LIN {X 0,Y 300.295,Z 456.079,A -85,B 0,C 180,E1 -16621.818,E2 -16621.818} C_VEL
LIN {X 0,Y 302.609,Z 468.728,A -85,B 0,C 180,E1 -16623.149,E2 -16623.149} C_VEL
LIN {X 0,Y 303.712,Z 478.266,A -85,B 0,C 180,E1 -16624.27,E2 -16624.27} C_VEL
LIN {X 0,Y 301.679,Z 491.184,A -85,B 0,C 180,E1 -16625.757,E2 -16625.757} C_VEL
LIN {X 0,Y 299.382,Z 502.708,A -85,B 0,C 180,E1 -16627.393,E2 -16627.393} C_VEL
LIN {X 0,Y 297.232,Z 513.15,A -85,B 0,C 180,E1 -16629.226,E2 -16629.226} C_VEL
LIN {X 0,Y 295.179,Z 522.585,A -85,B 0,C 180,E1 -16631.251,E2 -16631.251} C_VEL
LIN {X 0,Y 293.39,Z 531.306,A -85,B 0,C 180,E1 -16633.567,E2 -16633.567} C_VEL
LIN {X 0,Y 291.879,Z 538.835,A -85,B 0,C 180,E1 -16636.067,E2 -16636.067} C_VEL
LIN {X 0,Y 290.836,Z 543.926,A -85,B 0,C 180,E1 -16638.147,E2 -16638.147} C_VEL
LIN {X 0,Y 290.013,Z 549.179,A -85,B 0,C 180,E1 -16640.937,E2 -16640.937} C_VEL
LIN {X 0,Y 289.605,Z 552.122,A -85,B 0,C 180,E1 -16643.031,E2 -16643.031} C_VEL
LIN {X 0,Y 289.393,Z 554.815,A -85,B 0,C 180,E1 -16645.822,E2 -16645.822} C_VEL
LIN {X 0,Y 289.37,Z 556.148,A -85,B 0,C 180,E1 -16648.608,E2 -16648.608} C_VEL
LIN {X 0,Y 289.37,Z 556.142,A -85,B 0,C 180,E1 -16651.392,E2 -16651.392} C_VEL
LIN {X 0,Y 289.394,Z 554.801,A -85,B 0,C 180,E1 -16654.178,E2 -16654.178} C_VEL
LIN {X 0,Y 289.635,Z 552.099,A -85,B 0,C 180,E1 -16656.968,E2 -16656.968} C_VEL
LIN {X 0,Y 290.155,Z 547.96,A -85,B 0,C 180,E1 -16659.762,E2 -16659.762} C_VEL
LIN {X 0,Y 291.096,Z 542.261,A -85,B 0,C 180,E1 -16662.55,E2 -16662.55} C_VEL
LIN {X 0,Y 292.455,Z 535.839,A -85,B 0,C 180,E1 -16664.971,E2 -16664.971} C_VEL
LIN {X 0,Y 294.069,Z 527.863,A -85,B 0,C 180,E1 -16667.381,E2 -16667.381} C_VEL
LIN {X 0,Y 295.831,Z 519.513,A -85,B 0,C 180,E1 -16669.426,E2 -16669.426} C_VEL
LIN {X 0,Y 298.01,Z 509.466,A -85,B 0,C 180,E1 -16671.441,E2 -16671.441} C_VEL
LIN {X 0,Y 300.3,Z 498.252,A -85,B 0,C 180,E1 -16673.262,E2 -16673.262} C_VEL
LIN {X 0,Y 302.354,Z 487.095,A -85,B 0,C 180,E1 -16674.733,E2 -16674.733} C_VEL
LIN {X 0,Y 303.612,Z 477.752,A -85,B 0,C 180,E1 -16675.774,E2 -16675.774} C_VEL
LIN {X 0,Y 302.073,Z 465.248,A -85,B 0,C 180,E1 -16677.202,E2 -16677.202} C_VEL
LIN {X 0,Y 299.462,Z 452.518,A -85,B 0,C 180,E1 -16678.499,E2 -16678.499} C_VEL
LIN {X 0,Y 295.713,Z 438.551,A -85,B 0,C 180,E1 -16679.75,E2 -16679.75} C_VEL
LIN {X 0,Y 291.433,Z 426.246,A -85,B 0,C 180,E1 -16680.738,E2 -16680.738} C_VEL
LIN {X 0,Y 291.338,Z 425.398,A -85,B 0,C 180,E1 -16680.838,E2 -16680.838} C_VEL
LIN {X 0,Y 291.981,Z 420.382,A -85,B 0,C 180,E1 -16685.287,E2 -16685.287} C_VEL
LIN {X 0,Y 292.367,Z 416.77,A -85,B 0,C 180,E1 -16688.682,E2 -16688.682} C_VEL
LIN {X 0,Y 292.333,Z 413.602,A -85,B 0,C 180,E1 -16691.818,E2 -16691.818} C_VEL
LIN {X 0,Y 291.868,Z 409.987,A -85,B 0,C 180,E1 -16695.709,E2 -16695.709} C_VEL
LIN {X 0,Y 291.385,Z 406.828,A -85,B 0,C 180,E1 -16699.366,E2 -16699.366} C_VEL
LIN {X 0,Y 291.434,Z 406.81,A -85,B 0,C 180,E1 -16702.924,E2 -16702.924} C_VEL
LIN {X 0,Y 291.345,Z 406.822,A -85,B 0,C 180,E1 -16706.302,E2 -16706.302} C_VEL
LIN {X 0,Y 291.384,Z 406.816,A -85,B 0,C 180,E1 -16710.261,E2 -16710.261} C_VEL
LIN {X 0,Y 291.416,Z 406.812,A -85,B 0,C 180,E1 -16714.272,E2 -16714.272} C_VEL
LIN {X 0,Y 291.375,Z 406.817,A -85,B 0,C 180,E1 -16717.299,E2 -16717.299} C_VEL
LIN {X 0,Y 291.458,Z 406.805,A -85,B 0,C 180,E1 -16720.27,E2 -16720.27} C_VEL
LIN {X 0,Y 291.556,Z 406.792,A -85,B 0,C 180,E1 -16724.624,E2 -16724.624} C_VEL
LIN {X 0,Y 291.538,Z 406.791,A -85,B 0,C 180,E1 -16728.881,E2 -16728.881} C_VEL
LIN {X 0,Y 291.711,Z 406.773,A -85,B 0,C 180,E1 -16731.689,E2 -16731.689} C_VEL
LIN {X 0,Y 291.633,Z 406.783,A -85,B 0,C 180,E1 -16734.468,E2 -16734.468} C_VEL
LIN {X 0,Y 291.892,Z 406.753,A -85,B 0,C 180,E1 -16738.62,E2 -16738.62} C_VEL
LIN {X 0,Y 291.891,Z 406.752,A -85,B 0,C 180,E1 -16741.38,E2 -16741.38} C_VEL
LIN {X 0,Y 291.748,Z 406.769,A -85,B 0,C 180,E1 -16746.918,E2 -16746.918} C_VEL
LIN {X 0,Y 291.631,Z 406.786,A -85,B 0,C 180,E1 -16749.712,E2 -16749.712} C_VEL
LIN {X 0,Y 291.523,Z 406.792,A -85,B 0,C 180,E1 -16753.95,E2 -16753.95} C_VEL
LIN {X 0,Y 291.489,Z 406.796,A -85,B 0,C 180,E1 -16756.818,E2 -16756.818} C_VEL
LIN {X 0,Y 291.452,Z 406.806,A -85,B 0,C 180,E1 -16759.875,E2 -16759.875} C_VEL
LIN {X 0,Y 291.401,Z 406.813,A -85,B 0,C 180,E1 -16764.205,E2 -16764.205} C_VEL
LIN {X 0,Y 291.422,Z 406.81,A -85,B 0,C 180,E1 -16767.272,E2 -16767.272} C_VEL
LIN {X 0,Y 291.335,Z 406.82,A -85,B 0,C 180,E1 -16770.437,E2 -16770.437} C_VEL
LIN {X 0,Y 291.346,Z 406.82,A -85,B 0,C 180,E1 -16773.698,E2 -16773.698} C_VEL
LIN {X 0,Y 291.396,Z 406.815,A -85,B 0,C 180,E1 -16777.259,E2 -16777.259} C_VEL
LIN {X 0,Y 291.335,Z 406.823,A -85,B 0,C 180,E1 -16780.642,E2 -16780.642} C_VEL
LIN {X 0,Y 291.328,Z 406.82,A -85,B 0,C 180,E1 -16783.637,E2 -16783.637} C_VEL
LIN {X 0,Y 291.766,Z 409.919,A -85,B 0,C 180,E1 -16787.588,E2 -16787.588} C_VEL
LIN {X 0,Y 291.906,Z 412.394,A -85,B 0,C 180,E1 -16790.394,E2 -16790.394} C_VEL
LIN {X 0,Y 291.817,Z 414.778,A -85,B 0,C 180,E1 -16792.98,E2 -16792.98} C_VEL
LIN {X 0,Y 291.499,Z 417.991,A -85,B 0,C 180,E1 -16796.322,E2 -16796.322} C_VEL
LIN {X 0,Y 291.169,Z 420.912,A -85,B 0,C 180,E1 -16799.241,E2 -16799.241} C_VEL
LIN {X 0,Y 292.268,Z 424.311,A -85,B 0,C 180,E1 -16799.502,E2 -16799.502} C_VEL
LIN {X 0,Y 297.035,Z 437.696,A -85,B 0,C 180,E1 -16800.662,E2 -16800.662} C_VEL
LIN {X 0,Y 300.646,Z 451.139,A -85,B 0,C 180,E1 -16801.942,E2 -16801.942} C_VEL
LIN {X 0,Y 303.006,Z 462.696,A -85,B 0,C 180,E1 -16803.185,E2 -16803.185} C_VEL
LIN {X 0,Y 304.162,Z 470.973,A -85,B 0,C 180,E1 -16804.15,E2 -16804.15} C_VEL
LIN {X 0,Y 302.788,Z 481.413,A -85,B 0,C 180,E1 -16805.305,E2 -16805.305} C_VEL
LIN {X 0,Y 300.717,Z 492.606,A -85,B 0,C 180,E1 -16806.773,E2 -16806.773} C_VEL
LIN {X 0,Y 298.355,Z 503.859,A -85,B 0,C 180,E1 -16808.585,E2 -16808.585} C_VEL
LIN {X 0,Y 296.208,Z 513.912,A -85,B 0,C 180,E1 -16810.599,E2 -16810.599} C_VEL
LIN {X 0,Y 294.184,Z 523.069,A -85,B 0,C 180,E1 -16812.862,E2 -16812.862} C_VEL
LIN {X 0,Y 292.864,Z 530.227,A -85,B 0,C 180,E1 -16815.05,E2 -16815.05} C_VEL
LIN {X 0,Y 291.379,Z 536.643,A -85,B 0,C 180,E1 -16817.463,E2 -16817.463} C_VEL
LIN {X 0,Y 290.364,Z 542.331,A -85,B 0,C 180,E1 -16820.246,E2 -16820.246} C_VEL
LIN {X 0,Y 289.775,Z 546.463,A -85,B 0,C 180,E1 -16823.035,E2 -16823.035} C_VEL
LIN {X 0,Y 289.481,Z 549.164,A -85,B 0,C 180,E1 -16825.823,E2 -16825.823} C_VEL
LIN {X 0,Y 289.384,Z 550.516,A -85,B 0,C 180,E1 -16828.609,E2 -16828.609} C_VEL
LIN {X 0,Y 289.383,Z 550.546,A -85,B 0,C 180,E1 -16831.392,E2 -16831.392} C_VEL
LIN {X 0,Y 289.48,Z 549.251,A -85,B 0,C 180,E1 -16834.177,E2 -16834.177} C_VEL
LIN {X 0,Y 289.774,Z 546.601,A -85,B 0,C 180,E1 -16836.965,E2 -16836.965} C_VEL
LIN {X 0,Y 290.348,Z 542.528,A -85,B 0,C 180,E1 -16839.755,E2 -16839.755} C_VEL
LIN {X 0,Y 291.351,Z 536.901,A -85,B 0,C 180,E1 -16842.539,E2 -16842.539} C_VEL
LIN {X 0,Y 292.822,Z 530.546,A -85,B 0,C 180,E1 -16844.952,E2 -16844.952} C_VEL
LIN {X 0,Y 294.402,Z 522.572,A -85,B 0,C 180,E1 -16847.384,E2 -16847.384} C_VEL
LIN {X 0,Y 296.171,Z 514.38,A -85,B 0,C 180,E1 -16849.403,E2 -16849.403} C_VEL
LIN {X 0,Y 298.315,Z 504.42,A -85,B 0,C 180,E1 -16851.418,E2 -16851.418} C_VEL
LIN {X 0,Y 300.625,Z 493.329,A -85,B 0,C 180,E1 -16853.235,E2 -16853.235} C_VEL
LIN {X 0,Y 302.888,Z 480.905,A -85,B 0,C 180,E1 -16854.867,E2 -16854.867} C_VEL
LIN {X 0,Y 304.238,Z 471.314,A -85,B 0,C 180,E1 -16855.918,E2 -16855.918} C_VEL
LIN {X 0,Y 302.444,Z 459.661,A -85,B 0,C 180,E1 -16857.273,E2 -16857.273} C_VEL
LIN {X 0,Y 299.411,Z 446.078,A -85,B 0,C 180,E1 -16858.677,E2 -16858.677} C_VEL
LIN {X 0,Y 295.835,Z 433.958,A -85,B 0,C 180,E1 -16859.791,E2 -16859.791} C_VEL
LIN {X 0,Y 291.248,Z 421.639,A -85,B 0,C 180,E1 -16860.828,E2 -16860.828} C_VEL
LIN {X 0,Y 291.129,Z 420.907,A -85,B 0,C 180,E1 -16860.89,E2 -16860.89} C_VEL
LIN {X 0,Y 291.653,Z 416.829,A -85,B 0,C 180,E1 -16864.985,E2 -16864.985} C_VEL
LIN {X 0,Y 291.882,Z 413.257,A -85,B 0,C 180,E1 -16868.758,E2 -16868.758} C_VEL
LIN {X 0,Y 291.856,Z 410.636,A -85,B 0,C 180,E1 -16871.712,E2 -16871.712} C_VEL
LIN {X 0,Y 291.416,Z 407.395,A -85,B 0,C 180,E1 -16875.622,E2 -16875.622} C_VEL
LIN {X 0,Y 291.337,Z 406.828,A -85,B 0,C 180,E1 -16876.361,E2 -16876.361} C_VEL
LIN {X 0,Y 291.383,Z 406.815,A -85,B 0,C 180,E1 -16880.518,E2 -16880.518} C_VEL
LIN {X 0,Y 291.41,Z 406.813,A -85,B 0,C 180,E1 -16882.92,E2 -16882.92} C_VEL
LIN {X 0,Y 291.347,Z 406.82,A -85,B 0,C 180,E1 -16886.302,E2 -16886.302} C_VEL
LIN {X 0,Y 291.389,Z 406.812,A -85,B 0,C 180,E1 -16890.26,E2 -16890.26} C_VEL
LIN {X 0,Y 291.419,Z 406.811,A -85,B 0,C 180,E1 -16894.272,E2 -16894.272} C_VEL
LIN {X 0,Y 291.384,Z 406.814,A -85,B 0,C 180,E1 -16897.3,E2 -16897.3} C_VEL
LIN {X 0,Y 291.461,Z 406.8,A -85,B 0,C 180,E1 -16900.27,E2 -16900.27} C_VEL
LIN {X 0,Y 291.558,Z 406.791,A -85,B 0,C 180,E1 -16904.624,E2 -16904.624} C_VEL
LIN {X 0,Y 291.54,Z 406.795,A -85,B 0,C 180,E1 -16908.881,E2 -16908.881} C_VEL
LIN {X 0,Y 291.712,Z 406.772,A -85,B 0,C 180,E1 -16911.688,E2 -16911.688} C_VEL
LIN {X 0,Y 291.634,Z 406.783,A -85,B 0,C 180,E1 -16914.468,E2 -16914.468} C_VEL
LIN {X 0,Y 291.601,Z 406.783,A -85,B 0,C 180,E1 -16916.223,E2 -16916.223} C_VEL
LIN {X 0,Y 291.077,Z 406.853,A -85,B 0,C 180,E1 -16917.379,E2 -16917.379} C_VEL
LIN {X 0,Y 288.348,Z 407.192,A -85,B 0,C 180,E1 -16919.264,E2 -16919.264} C_VEL
LIN {X 0,Y 285.936,Z 407.49,A -85,B 0,C 180,E1 -16920.794,E2 -16920.794} C_VEL
LIN {X 0,Y 284.866,Z 407.627,A -85,B 0,C 180,E1 -16921.978,E2 -16921.978} C_VEL
LIN {X 0,Y 284.764,Z 407.636,A -85,B 0,C 180,E1 -16922.379,E2 -16922.379} C_VEL
LIN {X 0,Y 284.701,Z 407.646,A -85,B 0,C 180,E1 -16927.09,E2 -16927.09} C_VEL
LIN {X 0,Y 284.569,Z 407.663,A -85,B 0,C 180,E1 -16929.955,E2 -16929.955} C_VEL
LIN {X 0,Y 284.484,Z 407.675,A -85,B 0,C 180,E1 -16934.303,E2 -16934.303} C_VEL
LIN {X 0,Y 284.428,Z 407.679,A -85,B 0,C 180,E1 -16937.248,E2 -16937.248} C_VEL
LIN {X 0,Y 284.381,Z 407.687,A -85,B 0,C 180,E1 -16940.242,E2 -16940.242} C_VEL
LIN {X 0,Y 284.371,Z 407.682,A -85,B 0,C 180,E1 -16943.875,E2 -16943.875} C_VEL
LIN {X 0,Y 284.397,Z 407.68,A -85,B 0,C 180,E1 -16947.173,E2 -16947.173} C_VEL
LIN {X 0,Y 284.296,Z 407.698,A -85,B 0,C 180,E1 -16951.274,E2 -16951.274} C_VEL
LIN {X 0,Y 284.364,Z 407.692,A -85,B 0,C 180,E1 -16955.354,E2 -16955.354} C_VEL
LIN {X 0,Y 284.336,Z 407.697,A -85,B 0,C 180,E1 -16958.165,E2 -16958.165} C_VEL
LIN {X 0,Y 284.353,Z 407.696,A -85,B 0,C 180,E1 -16959.987,E2 -16959.987} C_VEL
LIN {X 0,Y 284.834,Z 410.735,A -85,B 0,C 180,E1 -16963.699,E2 -16963.699} C_VEL
LIN {X 0,Y 285.3,Z 414.29,A -85,B 0,C 180,E1 -16967.647,E2 -16967.647} C_VEL
LIN {X 0,Y 285.408,Z 416.721,A -85,B 0,C 180,E1 -16970.19,E2 -16970.19} C_VEL
LIN {X 0,Y 285.08,Z 420.364,A -85,B 0,C 180,E1 -16973.724,E2 -16973.724} C_VEL
LIN {X 0,Y 284.462,Z 424.903,A -85,B 0,C 180,E1 -16977.913,E2 -16977.913} C_VEL
LIN {X 0,Y 284.389,Z 425.386,A -85,B 0,C 180,E1 -16978.347,E2 -16978.347} C_VEL
LIN {X 0,Y 285.345,Z 428.635,A -85,B 0,C 180,E1 -16978.584,E2 -16978.584} C_VEL
LIN {X 0,Y 290.093,Z 442.311,A -85,B 0,C 180,E1 -16979.792,E2 -16979.792} C_VEL
LIN {X 0,Y 293.548,Z 456.013,A -85,B 0,C 180,E1 -16981.11,E2 -16981.11} C_VEL
LIN {X 0,Y 295.849,Z 468.661,A -85,B 0,C 180,E1 -16982.484,E2 -16982.484} C_VEL
LIN {X 0,Y 297.074,Z 480.142,A -85,B 0,C 180,E1 -16983.883,E2 -16983.883} C_VEL
LIN {X 0,Y 294.967,Z 492.411,A -85,B 0,C 180,E1 -16985.357,E2 -16985.357} C_VEL
LIN {X 0,Y 292.608,Z 503.706,A -85,B 0,C 180,E1 -16987.027,E2 -16987.027} C_VEL
LIN {X 0,Y 290.195,Z 514.769,A -85,B 0,C 180,E1 -16989.07,E2 -16989.07} C_VEL
LIN {X 0,Y 288.107,Z 523.897,A -85,B 0,C 180,E1 -16991.142,E2 -16991.142} C_VEL
LIN {X 0,Y 286.528,Z 530.915,A -85,B 0,C 180,E1 -16993.057,E2 -16993.057} C_VEL
LIN {X 0,Y 285.382,Z 536.846,A -85,B 0,C 180,E1 -16995.014,E2 -16995.014} C_VEL
LIN {X 0,Y 284.142,Z 542.246,A -85,B 0,C 180,E1 -16997.138,E2 -16997.138} C_VEL
LIN {X 0,Y 283.145,Z 547.93,A -85,B 0,C 180,E1 -16999.994,E2 -16999.994} C_VEL
LIN {X 0,Y 282.552,Z 552.054,A -85,B 0,C 180,E1 -17002.856,E2 -17002.856} C_VEL
LIN {X 0,Y 282.304,Z 554.747,A -85,B 0,C 180,E1 -17005.717,E2 -17005.717} C_VEL
LIN {X 0,Y 282.295,Z 556.079,A -85,B 0,C 180,E1 -17008.573,E2 -17008.573} C_VEL
LIN {X 0,Y 282.295,Z 556.074,A -85,B 0,C 180,E1 -17011.426,E2 -17011.426} C_VEL
LIN {X 0,Y 282.305,Z 554.732,A -85,B 0,C 180,E1 -17014.283,E2 -17014.283} C_VEL
LIN {X 0,Y 282.572,Z 552.03,A -85,B 0,C 180,E1 -17017.144,E2 -17017.144} C_VEL
LIN {X 0,Y 283.131,Z 547.89,A -85,B 0,C 180,E1 -17020.006,E2 -17020.006} C_VEL
LIN {X 0,Y 284.14,Z 542.191,A -85,B 0,C 180,E1 -17022.862,E2 -17022.862} C_VEL
LIN {X 0,Y 285.528,Z 535.768,A -85,B 0,C 180,E1 -17025.343,E2 -17025.343} C_VEL
LIN {X 0,Y 287.248,Z 527.789,A -85,B 0,C 180,E1 -17027.808,E2 -17027.808} C_VEL
LIN {X 0,Y 289.127,Z 519.442,A -85,B 0,C 180,E1 -17029.895,E2 -17029.895} C_VEL
LIN {X 0,Y 291.365,Z 509.394,A -85,B 0,C 180,E1 -17031.955,E2 -17031.955} C_VEL
LIN {X 0,Y 293.767,Z 498.179,A -85,B 0,C 180,E1 -17033.81,E2 -17033.81} C_VEL
LIN {X 0,Y 295.899,Z 487.022,A -85,B 0,C 180,E1 -17035.31,E2 -17035.31} C_VEL
LIN {X 0,Y 297.035,Z 479.43,A -85,B 0,C 180,E1 -17036.179,E2 -17036.179} C_VEL
LIN {X 0,Y 295.657,Z 467.162,A -85,B 0,C 180,E1 -17037.651,E2 -17037.651} C_VEL
LIN {X 0,Y 292.984,Z 453.827,A -85,B 0,C 180,E1 -17039.084,E2 -17039.084} C_VEL
LIN {X 0,Y 289.542,Z 440.775,A -85,B 0,C 180,E1 -17040.323,E2 -17040.323} C_VEL
LIN {X 0,Y 285.13,Z 428.161,A -85,B 0,C 180,E1 -17041.425,E2 -17041.425} C_VEL
LIN {X 0,Y 284.377,Z 425.375,A -85,B 0,C 180,E1 -17041.628,E2 -17041.628} C_VEL
LIN {X 0,Y 284.981,Z 421.125,A -85,B 0,C 180,E1 -17045.529,E2 -17045.529} C_VEL
LIN {X 0,Y 285.289,Z 418.511,A -85,B 0,C 180,E1 -17048.015,E2 -17048.015} C_VEL
LIN {X 0,Y 285.387,Z 416.271,A -85,B 0,C 180,E1 -17050.234,E2 -17050.234} C_VEL
LIN {X 0,Y 285.14,Z 413.066,A -85,B 0,C 180,E1 -17053.641,E2 -17053.641} C_VEL
LIN {X 0,Y 284.628,Z 409.423,A -85,B 0,C 180,E1 -17057.796,E2 -17057.796} C_VEL
LIN {X 0,Y 284.352,Z 407.693,A -85,B 0,C 180,E1 -17060.013,E2 -17060.013} C_VEL
LIN {X 0,Y 284.356,Z 407.691,A -85,B 0,C 180,E1 -17063.618,E2 -17063.618} C_VEL
LIN {X 0,Y 284.308,Z 407.698,A -85,B 0,C 180,E1 -17067.19,E2 -17067.19} C_VEL
LIN {X 0,Y 284.356,Z 407.692,A -85,B 0,C 180,E1 -17070.376,E2 -17070.376} C_VEL
LIN {X 0,Y 284.378,Z 407.688,A -85,B 0,C 180,E1 -17073.587,E2 -17073.587} C_VEL
LIN {X 0,Y 284.334,Z 407.693,A -85,B 0,C 180,E1 -17076.704,E2 -17076.704} C_VEL
LIN {X 0,Y 284.404,Z 407.683,A -85,B 0,C 180,E1 -17081.262,E2 -17081.262} C_VEL
LIN {X 0,Y 284.493,Z 407.672,A -85,B 0,C 180,E1 -17084.459,E2 -17084.459} C_VEL
LIN {X 0,Y 284.49,Z 407.669,A -85,B 0,C 180,E1 -17088.602,E2 -17088.602} C_VEL
LIN {X 0,Y 284.661,Z 407.652,A -85,B 0,C 180,E1 -17091.481,E2 -17091.481} C_VEL
LIN {X 0,Y 284.603,Z 407.658,A -85,B 0,C 180,E1 -17094.331,E2 -17094.331} C_VEL
LIN {X 0,Y 284.857,Z 407.629,A -85,B 0,C 180,E1 -17098.586,E2 -17098.586} C_VEL
LIN {X 0,Y 284.857,Z 407.629,A -85,B 0,C 180,E1 -17101.414,E2 -17101.414} C_VEL
LIN {X 0,Y 284.7,Z 407.647,A -85,B 0,C 180,E1 -17107.09,E2 -17107.09} C_VEL
LIN {X 0,Y 284.568,Z 407.663,A -85,B 0,C 180,E1 -17109.955,E2 -17109.955} C_VEL
LIN {X 0,Y 284.483,Z 407.67,A -85,B 0,C 180,E1 -17114.303,E2 -17114.303} C_VEL
LIN {X 0,Y 284.427,Z 407.676,A -85,B 0,C 180,E1 -17117.248,E2 -17117.248} C_VEL
LIN {X 0,Y 284.38,Z 407.686,A -85,B 0,C 180,E1 -17120.242,E2 -17120.242} C_VEL
LIN {X 0,Y 284.37,Z 407.688,A -85,B 0,C 180,E1 -17123.876,E2 -17123.876} C_VEL
LIN {X 0,Y 284.397,Z 407.685,A -85,B 0,C 180,E1 -17127.173,E2 -17127.173} C_VEL
LIN {X 0,Y 284.295,Z 407.698,A -85,B 0,C 180,E1 -17131.275,E2 -17131.275} C_VEL
LIN {X 0,Y 284.363,Z 407.69,A -85,B 0,C 180,E1 -17135.354,E2 -17135.354} C_VEL
LIN {X 0,Y 284.324,Z 407.692,A -85,B 0,C 180,E1 -17138.167,E2 -17138.167} C_VEL
LIN {X 0,Y 284.27,Z 407.702,A -85,B 0,C 180,E1 -17142.125,E2 -17142.125} C_VEL
LIN {X 0,Y 284.375,Z 408.375,A -85,B 0,C 180,E1 -17144.217,E2 -17144.217} C_VEL
LIN {X 0,Y 284.86,Z 411.602,A -85,B 0,C 180,E1 -17148.23,E2 -17148.23} C_VEL
LIN {X 0,Y 284.83,Z 414.853,A -85,B 0,C 180,E1 -17151.913,E2 -17151.913} C_VEL
LIN {X 0,Y 284.558,Z 418.073,A -85,B 0,C 180,E1 -17155.386,E2 -17155.386} C_VEL
LIN {X 0,Y 284.227,Z 421.003,A -85,B 0,C 180,E1 -17158.416,E2 -17158.416} C_VEL
LIN {X 0,Y 285.22,Z 424.218,A -85,B 0,C 180,E1 -17158.658,E2 -17158.658} C_VEL
LIN {X 0,Y 290.073,Z 437.415,A -85,B 0,C 180,E1 -17159.865,E2 -17159.865} C_VEL
LIN {X 0,Y 293.876,Z 451.158,A -85,B 0,C 180,E1 -17161.231,E2 -17161.231} C_VEL
LIN {X 0,Y 296.453,Z 463.855,A -85,B 0,C 180,E1 -17162.647,E2 -17162.647} C_VEL
LIN {X 0,Y 297.595,Z 473.419,A -85,B 0,C 180,E1 -17163.82,E2 -17163.82} C_VEL
LIN {X 0,Y 295.605,Z 485.426,A -85,B 0,C 180,E1 -17165.227,E2 -17165.227} C_VEL
LIN {X 0,Y 293.256,Z 497.006,A -85,B 0,C 180,E1 -17166.894,E2 -17166.894} C_VEL
LIN {X 0,Y 291.005,Z 507.488,A -85,B 0,C 180,E1 -17168.761,E2 -17168.761} C_VEL
LIN {X 0,Y 288.832,Z 516.948,A -85,B 0,C 180,E1 -17170.823,E2 -17170.823} C_VEL
LIN {X 0,Y 286.817,Z 525.968,A -85,B 0,C 180,E1 -17173.267,E2 -17173.267} C_VEL
LIN {X 0,Y 285.733,Z 531.302,A -85,B 0,C 180,E1 -17175.033,E2 -17175.033} C_VEL
LIN {X 0,Y 284.416,Z 536.714,A -85,B 0,C 180,E1 -17177.151,E2 -17177.151} C_VEL
LIN {X 0,Y 283.351,Z 542.401,A -85,B 0,C 180,E1 -17180.002,E2 -17180.002} C_VEL
LIN {X 0,Y 282.726,Z 546.533,A -85,B 0,C 180,E1 -17182.86,E2 -17182.86} C_VEL
LIN {X 0,Y 282.392,Z 549.234,A -85,B 0,C 180,E1 -17185.718,E2 -17185.718} C_VEL
LIN {X 0,Y 282.309,Z 550.585,A -85,B 0,C 180,E1 -17188.574,E2 -17188.574} C_VEL
LIN {X 0,Y 282.309,Z 550.614,A -85,B 0,C 180,E1 -17191.427,E2 -17191.427} C_VEL
LIN {X 0,Y 282.391,Z 549.319,A -85,B 0,C 180,E1 -17194.282,E2 -17194.282} C_VEL
LIN {X 0,Y 282.726,Z 546.669,A -85,B 0,C 180,E1 -17197.14,E2 -17197.14} C_VEL
LIN {X 0,Y 283.333,Z 542.596,A -85,B 0,C 180,E1 -17199.999,E2 -17199.999} C_VEL
LIN {X 0,Y 284.389,Z 536.969,A -85,B 0,C 180,E1 -17202.851,E2 -17202.851} C_VEL
LIN {X 0,Y 285.947,Z 530.613,A -85,B 0,C 180,E1 -17205.32,E2 -17205.32} C_VEL
LIN {X 0,Y 287.581,Z 522.695,A -85,B 0,C 180,E1 -17207.793,E2 -17207.793} C_VEL
LIN {X 0,Y 289.449,Z 514.447,A -85,B 0,C 180,E1 -17209.873,E2 -17209.873} C_VEL
LIN {X 0,Y 291.718,Z 504.485,A -85,B 0,C 180,E1 -17211.927,E2 -17211.927} C_VEL
LIN {X 0,Y 294.1,Z 493.394,A -85,B 0,C 180,E1 -17213.782,E2 -17213.782} C_VEL
LIN {X 0,Y 296.22,Z 482.35,A -85,B 0,C 180,E1 -17215.281,E2 -17215.281} C_VEL
LIN {X 0,Y 297.691,Z 472.69,A -85,B 0,C 180,E1 -17216.375,E2 -17216.375} C_VEL
LIN {X 0,Y 295.938,Z 461.06,A -85,B 0,C 180,E1 -17217.795,E2 -17217.795} C_VEL
LIN {X 0,Y 293.151,Z 448.192,A -85,B 0,C 180,E1 -17219.193,E2 -17219.193} C_VEL
LIN {X 0,Y 289.954,Z 437.068,A -85,B 0,C 180,E1 -17220.29,E2 -17220.29} C_VEL
LIN {X 0,Y 284.966,Z 423.701,A -85,B 0,C 180,E1 -17221.515,E2 -17221.515} C_VEL
LIN {X 0,Y 284.222,Z 420.978,A -85,B 0,C 180,E1 -17221.732,E2 -17221.732} C_VEL
LIN {X 0,Y 284.65,Z 417.399,A -85,B 0,C 180,E1 -17225.435,E2 -17225.435} C_VEL
LIN {X 0,Y 284.83,Z 414.949,A -85,B 0,C 180,E1 -17228.087,E2 -17228.087} C_VEL
LIN {X 0,Y 284.9,Z 413.145,A -85,B 0,C 180,E1 -17230.118,E2 -17230.118} C_VEL
LIN {X 0,Y 284.794,Z 411.328,A -85,B 0,C 180,E1 -17232.241,E2 -17232.241} C_VEL
LIN {X 0,Y 284.354,Z 408.153,A -85,B 0,C 180,E1 -17236.208,E2 -17236.208} C_VEL
LIN {X 0,Y 284.274,Z 407.705,A -85,B 0,C 180,E1 -17238.125,E2 -17238.125} C_VEL
LIN {X 0,Y 284.325,Z 407.693,A -85,B 0,C 180,E1 -17242.278,E2 -17242.278} C_VEL
LIN {X 0,Y 284.311,Z 407.696,A -85,B 0,C 180,E1 -17245.351,E2 -17245.351} C_VEL
LIN {X 0,Y 284.298,Z 407.696,A -85,B 0,C 180,E1 -17248.726,E2 -17248.726} C_VEL
LIN {X 0,Y 284.4,Z 407.686,A -85,B 0,C 180,E1 -17252.826,E2 -17252.826} C_VEL
LIN {X 0,Y 284.369,Z 407.684,A -85,B 0,C 180,E1 -17256.707,E2 -17256.707} C_VEL
LIN {X 0,Y 284.407,Z 407.683,A -85,B 0,C 180,E1 -17261.262,E2 -17261.262} C_VEL
LIN {X 0,Y 284.495,Z 407.671,A -85,B 0,C 180,E1 -17264.459,E2 -17264.459} C_VEL
LIN {X 0,Y 284.491,Z 407.673,A -85,B 0,C 180,E1 -17268.601,E2 -17268.601} C_VEL
LIN {X 0,Y 284.662,Z 407.65,A -85,B 0,C 180,E1 -17271.481,E2 -17271.481} C_VEL
LIN {X 0,Y 284.604,Z 407.658,A -85,B 0,C 180,E1 -17274.331,E2 -17274.331} C_VEL
LIN {X 0,Y 284.857,Z 407.627,A -85,B 0,C 180,E1 -17278.586,E2 -17278.586} C_VEL
LIN {X 0,Y 284.859,Z 407.626,A -85,B 0,C 180,E1 -17281.414,E2 -17281.414} C_VEL
LIN {X 0,Y 284.764,Z 407.636,A -85,B 0,C 180,E1 -17282.379,E2 -17282.379} C_VEL
LIN {X 0,Y 284.044,Z 407.729,A -85,B 0,C 180,E1 -17283.558,E2 -17283.558} C_VEL
LIN {X 0,Y 281.132,Z 408.089,A -85,B 0,C 180,E1 -17285.478,E2 -17285.478} C_VEL
LIN {X 0,Y 278.703,Z 408.394,A -85,B 0,C 180,E1 -17287.036,E2 -17287.036} C_VEL
LIN {X 0,Y 277.686,Z 408.52,A -85,B 0,C 180,E1 -17288.245,E2 -17288.245} C_VEL
LIN {X 0,Y 277.616,Z 408.529,A -85,B 0,C 180,E1 -17288.655,E2 -17288.655} C_VEL
LIN {X 0,Y 277.42,Z 408.555,A -85,B 0,C 180,E1 -17293.179,E2 -17293.179} C_VEL
LIN {X 0,Y 277.409,Z 408.557,A -85,B 0,C 180,E1 -17296.181,E2 -17296.181} C_VEL
LIN {X 0,Y 277.347,Z 408.563,A -85,B 0,C 180,E1 -17300.35,E2 -17300.35} C_VEL
LIN {X 0,Y 277.321,Z 408.56,A -85,B 0,C 180,E1 -17304.17,E2 -17304.17} C_VEL
LIN {X 0,Y 277.325,Z 408.561,A -85,B 0,C 180,E1 -17307.504,E2 -17307.504} C_VEL
LIN {X 0,Y 277.274,Z 408.569,A -85,B 0,C 180,E1 -17310.481,E2 -17310.481} C_VEL
LIN {X 0,Y 277.256,Z 408.577,A -85,B 0,C 180,E1 -17313.894,E2 -17313.894} C_VEL
LIN {X 0,Y 277.292,Z 408.575,A -85,B 0,C 180,E1 -17317.465,E2 -17317.465} C_VEL
LIN {X 0,Y 277.269,Z 408.578,A -85,B 0,C 180,E1 -17319.322,E2 -17319.322} C_VEL
LIN {X 0,Y 277.761,Z 411.472,A -85,B 0,C 180,E1 -17323.091,E2 -17323.091} C_VEL
LIN {X 0,Y 278.237,Z 414.928,A -85,B 0,C 180,E1 -17327.097,E2 -17327.097} C_VEL
LIN {X 0,Y 278.352,Z 416.929,A -85,B 0,C 180,E1 -17329.24,E2 -17329.24} C_VEL
LIN {X 0,Y 278.153,Z 420.281,A -85,B 0,C 180,E1 -17332.67,E2 -17332.67} C_VEL
LIN {X 0,Y 277.647,Z 423.925,A -85,B 0,C 180,E1 -17336.159,E2 -17336.159} C_VEL
LIN {X 0,Y 277.48,Z 425.306,A -85,B 0,C 180,E1 -17337.457,E2 -17337.457} C_VEL
LIN {X 0,Y 278.453,Z 428.552,A -85,B 0,C 180,E1 -17337.712,E2 -17337.712} C_VEL
LIN {X 0,Y 282.652,Z 440.529,A -85,B 0,C 180,E1 -17338.813,E2 -17338.813} C_VEL
LIN {X 0,Y 285.635,Z 451.022,A -85,B 0,C 180,E1 -17339.847,E2 -17339.847} C_VEL
LIN {X 0,Y 288.458,Z 464.356,A -85,B 0,C 180,E1 -17341.295,E2 -17341.295} C_VEL
LIN {X 0,Y 290.007,Z 475.033,A -85,B 0,C 180,E1 -17342.584,E2 -17342.584} C_VEL
LIN {X 0,Y 290.497,Z 481.435,A -85,B 0,C 180,E1 -17343.413,E2 -17343.413} C_VEL
LIN {X 0,Y 288.267,Z 493.58,A -85,B 0,C 180,E1 -17344.937,E2 -17344.937} C_VEL
LIN {X 0,Y 286.053,Z 503.64,A -85,B 0,C 180,E1 -17346.469,E2 -17346.469} C_VEL
LIN {X 0,Y 283.537,Z 514.702,A -85,B 0,C 180,E1 -17348.555,E2 -17348.555} C_VEL
LIN {X 0,Y 281.374,Z 523.83,A -85,B 0,C 180,E1 -17350.673,E2 -17350.673} C_VEL
LIN {X 0,Y 279.419,Z 532.291,A -85,B 0,C 180,E1 -17353.098,E2 -17353.098} C_VEL
LIN {X 0,Y 278.063,Z 538.7,A -85,B 0,C 180,E1 -17355.36,E2 -17355.36} C_VEL
LIN {X 0,Y 276.567,Z 545.225,A -85,B 0,C 180,E1 -17358.27,E2 -17358.27} C_VEL
LIN {X 0,Y 275.761,Z 550.11,A -85,B 0,C 180,E1 -17361.204,E2 -17361.204} C_VEL
LIN {X 0,Y 275.3,Z 553.505,A -85,B 0,C 180,E1 -17364.139,E2 -17364.139} C_VEL
LIN {X 0,Y 275.21,Z 555.513,A -85,B 0,C 180,E1 -17367.072,E2 -17367.072} C_VEL
LIN {X 0,Y 275.218,Z 556.174,A -85,B 0,C 180,E1 -17370,E2 -17370} C_VEL
LIN {X 0,Y 275.211,Z 555.501,A -85,B 0,C 180,E1 -17372.927,E2 -17372.927} C_VEL
LIN {X 0,Y 275.335,Z 553.485,A -85,B 0,C 180,E1 -17375.86,E2 -17375.86} C_VEL
LIN {X 0,Y 275.763,Z 550.076,A -85,B 0,C 180,E1 -17378.796,E2 -17378.796} C_VEL
LIN {X 0,Y 276.562,Z 545.174,A -85,B 0,C 180,E1 -17381.73,E2 -17381.73} C_VEL
LIN {X 0,Y 278.061,Z 538.636,A -85,B 0,C 180,E1 -17384.64,E2 -17384.64} C_VEL
LIN {X 0,Y 279.642,Z 531.138,A -85,B 0,C 180,E1 -17387.25,E2 -17387.25} C_VEL
LIN {X 0,Y 281.697,Z 522.346,A -85,B 0,C 180,E1 -17389.682,E2 -17389.682} C_VEL
LIN {X 0,Y 283.964,Z 512.89,A -85,B 0,C 180,E1 -17391.792,E2 -17391.792} C_VEL
LIN {X 0,Y 286.304,Z 502.42,A -85,B 0,C 180,E1 -17393.701,E2 -17393.701} C_VEL
LIN {X 0,Y 288.756,Z 490.865,A -85,B 0,C 180,E1 -17395.402,E2 -17395.402} C_VEL
LIN {X 0,Y 290.443,Z 481.211,A -85,B 0,C 180,E1 -17396.592,E2 -17396.592} C_VEL
LIN {X 0,Y 289.328,Z 469.598,A -85,B 0,C 180,E1 -17398.058,E2 -17398.058} C_VEL
LIN {X 0,Y 286.847,Z 456.37,A -85,B 0,C 180,E1 -17399.565,E2 -17399.565} C_VEL
LIN {X 0,Y 283.415,Z 442.904,A -85,B 0,C 180,E1 -17400.926,E2 -17400.926} C_VEL
LIN {X 0,Y 278.675,Z 428.985,A -85,B 0,C 180,E1 -17402.207,E2 -17402.207} C_VEL
LIN {X 0,Y 277.534,Z 425.945,A -85,B 0,C 180,E1 -17402.464,E2 -17402.464} C_VEL
LIN {X 0,Y 277.461,Z 425.247,A -85,B 0,C 180,E1 -17402.566,E2 -17402.566} C_VEL
LIN {X 0,Y 278.024,Z 421.603,A -85,B 0,C 180,E1 -17406.011,E2 -17406.011} C_VEL
LIN {X 0,Y 278.315,Z 418.438,A -85,B 0,C 180,E1 -17409.146,E2 -17409.146} C_VEL
LIN {X 0,Y 278.333,Z 416.634,A -85,B 0,C 180,E1 -17411.034,E2 -17411.034} C_VEL
LIN {X 0,Y 278.201,Z 414.806,A -85,B 0,C 180,E1 -17413.006,E2 -17413.006} C_VEL
LIN {X 0,Y 277.719,Z 411.174,A -85,B 0,C 180,E1 -17417.212,E2 -17417.212} C_VEL
LIN {X 0,Y 277.268,Z 408.574,A -85,B 0,C 180,E1 -17420.678,E2 -17420.678} C_VEL
LIN {X 0,Y 277.306,Z 408.57,A -85,B 0,C 180,E1 -17424.345,E2 -17424.345} C_VEL
LIN {X 0,Y 277.244,Z 408.578,A -85,B 0,C 180,E1 -17427.836,E2 -17427.836} C_VEL
LIN {X 0,Y 277.269,Z 408.574,A -85,B 0,C 180,E1 -17431.21,E2 -17431.21} C_VEL
LIN {X 0,Y 277.31,Z 408.569,A -85,B 0,C 180,E1 -17434.479,E2 -17434.479} C_VEL
LIN {X 0,Y 277.269,Z 408.573,A -85,B 0,C 180,E1 -17437.654,E2 -17437.654} C_VEL
LIN {X 0,Y 277.346,Z 408.564,A -85,B 0,C 180,E1 -17440.766,E2 -17440.766} C_VEL
LIN {X 0,Y 277.436,Z 408.548,A -85,B 0,C 180,E1 -17445.326,E2 -17445.326} C_VEL
LIN {X 0,Y 277.508,Z 408.539,A -85,B 0,C 180,E1 -17449.789,E2 -17449.789} C_VEL
LIN {X 0,Y 277.655,Z 408.518,A -85,B 0,C 180,E1 -17452.729,E2 -17452.729} C_VEL
LIN {X 0,Y 277.823,Z 408.505,A -85,B 0,C 180,E1 -17458.551,E2 -17458.551} C_VEL
LIN {X 0,Y 277.823,Z 408.505,A -85,B 0,C 180,E1 -17461.45,E2 -17461.45} C_VEL
LIN {X 0,Y 277.655,Z 408.524,A -85,B 0,C 180,E1 -17467.271,E2 -17467.271} C_VEL
LIN {X 0,Y 277.508,Z 408.542,A -85,B 0,C 180,E1 -17470.211,E2 -17470.211} C_VEL
LIN {X 0,Y 277.436,Z 408.551,A -85,B 0,C 180,E1 -17474.674,E2 -17474.674} C_VEL
LIN {X 0,Y 277.347,Z 408.564,A -85,B 0,C 180,E1 -17479.234,E2 -17479.234} C_VEL
LIN {X 0,Y 277.321,Z 408.567,A -85,B 0,C 180,E1 -17484.171,E2 -17484.171} C_VEL
LIN {X 0,Y 277.326,Z 408.566,A -85,B 0,C 180,E1 -17487.505,E2 -17487.505} C_VEL
LIN {X 0,Y 277.273,Z 408.572,A -85,B 0,C 180,E1 -17490.481,E2 -17490.481} C_VEL
LIN {X 0,Y 277.255,Z 408.575,A -85,B 0,C 180,E1 -17493.895,E2 -17493.895} C_VEL
LIN {X 0,Y 277.283,Z 408.572,A -85,B 0,C 180,E1 -17497.467,E2 -17497.467} C_VEL
LIN {X 0,Y 277.211,Z 408.58,A -85,B 0,C 180,E1 -17501.237,E2 -17501.237} C_VEL
LIN {X 0,Y 277.256,Z 408.824,A -85,B 0,C 180,E1 -17503.189,E2 -17503.189} C_VEL
LIN {X 0,Y 277.708,Z 411.939,A -85,B 0,C 180,E1 -17507.215,E2 -17507.215} C_VEL
LIN {X 0,Y 277.852,Z 413.697,A -85,B 0,C 180,E1 -17509.361,E2 -17509.361} C_VEL
LIN {X 0,Y 277.741,Z 416.532,A -85,B 0,C 180,E1 -17512.606,E2 -17512.606} C_VEL
LIN {X 0,Y 277.416,Z 419.765,A -85,B 0,C 180,E1 -17516.128,E2 -17516.128} C_VEL
LIN {X 0,Y 277.314,Z 421.121,A -85,B 0,C 180,E1 -17517.543,E2 -17517.543} C_VEL
LIN {X 0,Y 278.368,Z 424.339,A -85,B 0,C 180,E1 -17517.795,E2 -17517.795} C_VEL
LIN {X 0,Y 283.536,Z 438.347,A -85,B 0,C 180,E1 -17519.143,E2 -17519.143} C_VEL
LIN {X 0,Y 286.929,Z 450.464,A -85,B 0,C 180,E1 -17520.406,E2 -17520.406} C_VEL
LIN {X 0,Y 289.755,Z 463.935,A -85,B 0,C 180,E1 -17521.96,E2 -17521.96} C_VEL
LIN {X 0,Y 291.079,Z 474.396,A -85,B 0,C 180,E1 -17523.298,E2 -17523.298} C_VEL
LIN {X 0,Y 288.925,Z 486.788,A -85,B 0,C 180,E1 -17524.806,E2 -17524.806} C_VEL
LIN {X 0,Y 286.492,Z 498.146,A -85,B 0,C 180,E1 -17526.507,E2 -17526.507} C_VEL
LIN {X 0,Y 284.384,Z 507.56,A -85,B 0,C 180,E1 -17528.242,E2 -17528.242} C_VEL
LIN {X 0,Y 282.111,Z 517.019,A -85,B 0,C 180,E1 -17530.348,E2 -17530.348} C_VEL
LIN {X 0,Y 279.984,Z 526.04,A -85,B 0,C 180,E1 -17532.846,E2 -17532.846} C_VEL
LIN {X 0,Y 278.865,Z 531.373,A -85,B 0,C 180,E1 -17534.656,E2 -17534.656} C_VEL
LIN {X 0,Y 277.464,Z 536.785,A -85,B 0,C 180,E1 -17536.823,E2 -17536.823} C_VEL
LIN {X 0,Y 276.336,Z 542.471,A -85,B 0,C 180,E1 -17539.745,E2 -17539.745} C_VEL
LIN {X 0,Y 275.675,Z 546.602,A -85,B 0,C 180,E1 -17542.677,E2 -17542.677} C_VEL
LIN {X 0,Y 275.305,Z 549.303,A -85,B 0,C 180,E1 -17545.608,E2 -17545.608} C_VEL
LIN {X 0,Y 275.236,Z 550.654,A -85,B 0,C 180,E1 -17548.537,E2 -17548.537} C_VEL
LIN {X 0,Y 275.236,Z 550.683,A -85,B 0,C 180,E1 -17551.463,E2 -17551.463} C_VEL
LIN {X 0,Y 275.306,Z 549.388,A -85,B 0,C 180,E1 -17554.392,E2 -17554.392} C_VEL
LIN {X 0,Y 275.649,Z 546.737,A -85,B 0,C 180,E1 -17557.324,E2 -17557.324} C_VEL
LIN {X 0,Y 276.302,Z 542.664,A -85,B 0,C 180,E1 -17560.256,E2 -17560.256} C_VEL
LIN {X 0,Y 277.436,Z 537.037,A -85,B 0,C 180,E1 -17563.179,E2 -17563.179} C_VEL
LIN {X 0,Y 279.072,Z 530.68,A -85,B 0,C 180,E1 -17565.707,E2 -17565.707} C_VEL
LIN {X 0,Y 280.733,Z 523.026,A -85,B 0,C 180,E1 -17568.161,E2 -17568.161} C_VEL
LIN {X 0,Y 282.766,Z 514.513,A -85,B 0,C 180,E1 -17570.363,E2 -17570.363} C_VEL
LIN {X 0,Y 285.142,Z 504.551,A -85,B 0,C 180,E1 -17572.46,E2 -17572.46} C_VEL
LIN {X 0,Y 287.581,Z 493.459,A -85,B 0,C 180,E1 -17574.356,E2 -17574.356} C_VEL
LIN {X 0,Y 289.806,Z 482.414,A -85,B 0,C 180,E1 -17575.882,E2 -17575.882} C_VEL
LIN {X 0,Y 291.11,Z 473.868,A -85,B 0,C 180,E1 -17576.882,E2 -17576.882} C_VEL
LIN {X 0,Y 289.46,Z 462.451,A -85,B 0,C 180,E1 -17578.34,E2 -17578.34} C_VEL
LIN {X 0,Y 286.795,Z 449.935,A -85,B 0,C 180,E1 -17579.774,E2 -17579.774} C_VEL
LIN {X 0,Y 283.844,Z 439.424,A -85,B 0,C 180,E1 -17580.879,E2 -17580.879} C_VEL
LIN {X 0,Y 278.598,Z 424.716,A -85,B 0,C 180,E1 -17582.288,E2 -17582.288} C_VEL
LIN {X 0,Y 277.366,Z 421.604,A -85,B 0,C 180,E1 -17582.56,E2 -17582.56} C_VEL
LIN {X 0,Y 277.311,Z 421.051,A -85,B 0,C 180,E1 -17582.62,E2 -17582.62} C_VEL
LIN {X 0,Y 277.641,Z 417.986,A -85,B 0,C 180,E1 -17585.901,E2 -17585.901} C_VEL
LIN {X 0,Y 277.839,Z 415.022,A -85,B 0,C 180,E1 -17589.226,E2 -17589.226} C_VEL
LIN {X 0,Y 277.722,Z 412.033,A -85,B 0,C 180,E1 -17592.788,E2 -17592.788} C_VEL
LIN {X 0,Y 277.264,Z 408.938,A -85,B 0,C 180,E1 -17596.812,E2 -17596.812} C_VEL
LIN {X 0,Y 277.221,Z 408.585,A -85,B 0,C 180,E1 -17597.324,E2 -17597.324} C_VEL
LIN {X 0,Y 277.267,Z 408.572,A -85,B 0,C 180,E1 -17601.792,E2 -17601.792} C_VEL
LIN {X 0,Y 277.287,Z 408.571,A -85,B 0,C 180,E1 -17604.342,E2 -17604.342} C_VEL
LIN {X 0,Y 277.247,Z 408.574,A -85,B 0,C 180,E1 -17607.837,E2 -17607.837} C_VEL
LIN {X 0,Y 277.292,Z 408.57,A -85,B 0,C 180,E1 -17611.213,E2 -17611.213} C_VEL
LIN {X 0,Y 277.316,Z 408.568,A -85,B 0,C 180,E1 -17614.48,E2 -17614.48} C_VEL
LIN {X 0,Y 277.288,Z 408.571,A -85,B 0,C 180,E1 -17617.655,E2 -17617.655} C_VEL
LIN {X 0,Y 277.348,Z 408.562,A -85,B 0,C 180,E1 -17620.766,E2 -17620.766} C_VEL
LIN {X 0,Y 277.437,Z 408.552,A -85,B 0,C 180,E1 -17625.326,E2 -17625.326} C_VEL
LIN {X 0,Y 277.509,Z 408.542,A -85,B 0,C 180,E1 -17629.789,E2 -17629.789} C_VEL
LIN {X 0,Y 277.656,Z 408.524,A -85,B 0,C 180,E1 -17632.729,E2 -17632.729} C_VEL
LIN {X 0,Y 277.823,Z 408.503,A -85,B 0,C 180,E1 -17638.55,E2 -17638.55} C_VEL
LIN {X 0,Y 277.825,Z 408.502,A -85,B 0,C 180,E1 -17641.449,E2 -17641.449} C_VEL
LIN {X 0,Y 277.656,Z 408.524,A -85,B 0,C 180,E1 -17647.271,E2 -17647.271} C_VEL
LIN {X 0,Y 277.616,Z 408.529,A -85,B 0,C 180,E1 -17648.655,E2 -17648.655} C_VEL
LIN {X 0,Y 276.973,Z 408.616,A -85,B 0,C 180,E1 -17649.863,E2 -17649.863} C_VEL
LIN {X 0,Y 274.094,Z 408.977,A -85,B 0,C 180,E1 -17651.83,E2 -17651.83} C_VEL
LIN {X 0,Y 271.609,Z 409.283,A -85,B 0,C 180,E1 -17653.429,E2 -17653.429} C_VEL
LIN {X 0,Y 270.509,Z 409.416,A -85,B 0,C 180,E1 -17654.669,E2 -17654.669} C_VEL
LIN {X 0,Y 270.404,Z 409.427,A -85,B 0,C 180,E1 -17655.09,E2 -17655.09} C_VEL
LIN {X 0,Y 270.304,Z 409.442,A -85,B 0,C 180,E1 -17659.755,E2 -17659.755} C_VEL
LIN {X 0,Y 270.276,Z 409.439,A -85,B 0,C 180,E1 -17664.585,E2 -17664.585} C_VEL
LIN {X 0,Y 270.273,Z 409.441,A -85,B 0,C 180,E1 -17667.908,E2 -17667.908} C_VEL
LIN {X 0,Y 270.186,Z 409.456,A -85,B 0,C 180,E1 -17671.348,E2 -17671.348} C_VEL
LIN {X 0,Y 270.218,Z 409.453,A -85,B 0,C 180,E1 -17674.903,E2 -17674.903} C_VEL
LIN {X 0,Y 270.224,Z 409.455,A -85,B 0,C 180,E1 -17678.717,E2 -17678.717} C_VEL
LIN {X 0,Y 270.684,Z 412.203,A -85,B 0,C 180,E1 -17682.459,E2 -17682.459} C_VEL
LIN {X 0,Y 271.162,Z 415.604,A -85,B 0,C 180,E1 -17686.528,E2 -17686.528} C_VEL
LIN {X 0,Y 271.312,Z 418.408,A -85,B 0,C 180,E1 -17689.639,E2 -17689.639} C_VEL
LIN {X 0,Y 271.244,Z 420.233,A -85,B 0,C 180,E1 -17691.549,E2 -17691.549} C_VEL
LIN {X 0,Y 271.036,Z 422.138,A -85,B 0,C 180,E1 -17693.498,E2 -17693.498} C_VEL
LIN {X 0,Y 270.586,Z 425.24,A -85,B 0,C 180,E1 -17696.53,E2 -17696.53} C_VEL
LIN {X 0,Y 271.452,Z 428.255,A -85,B 0,C 180,E1 -17696.765,E2 -17696.765} C_VEL
LIN {X 0,Y 276.235,Z 441.502,A -85,B 0,C 180,E1 -17698.064,E2 -17698.064} C_VEL
LIN {X 0,Y 279.559,Z 453.724,A -85,B 0,C 180,E1 -17699.343,E2 -17699.343} C_VEL
LIN {X 0,Y 281.998,Z 465.751,A -85,B 0,C 180,E1 -17700.724,E2 -17700.724} C_VEL
LIN {X 0,Y 283.53,Z 476.768,A -85,B 0,C 180,E1 -17702.124,E2 -17702.124} C_VEL
LIN {X 0,Y 283.935,Z 481.953,A -85,B 0,C 180,E1 -17702.827,E2 -17702.827} C_VEL
LIN {X 0,Y 281.548,Z 494.765,A -85,B 0,C 180,E1 -17704.507,E2 -17704.507} C_VEL
LIN {X 0,Y 279.054,Z 505.54,A -85,B 0,C 180,E1 -17706.236,E2 -17706.236} C_VEL
LIN {X 0,Y 276.53,Z 516.265,A -85,B 0,C 180,E1 -17708.376,E2 -17708.376} C_VEL
LIN {X 0,Y 274.293,Z 525.119,A -85,B 0,C 180,E1 -17710.543,E2 -17710.543} C_VEL
LIN {X 0,Y 272.465,Z 532.733,A -85,B 0,C 180,E1 -17712.829,E2 -17712.829} C_VEL
LIN {X 0,Y 270.697,Z 540.445,A -85,B 0,C 180,E1 -17715.721,E2 -17715.721} C_VEL
LIN {X 0,Y 269.568,Z 545.156,A -85,B 0,C 180,E1 -17717.961,E2 -17717.961} C_VEL
LIN {X 0,Y 268.714,Z 550.041,A -85,B 0,C 180,E1 -17720.971,E2 -17720.971} C_VEL
LIN {X 0,Y 268.224,Z 553.436,A -85,B 0,C 180,E1 -17723.984,E2 -17723.984} C_VEL
LIN {X 0,Y 268.107,Z 555.444,A -85,B 0,C 180,E1 -17726.995,E2 -17726.995} C_VEL
LIN {X 0,Y 268.144,Z 556.106,A -85,B 0,C 180,E1 -17730,E2 -17730} C_VEL
LIN {X 0,Y 268.107,Z 555.432,A -85,B 0,C 180,E1 -17733.005,E2 -17733.005} C_VEL
LIN {X 0,Y 268.245,Z 553.415,A -85,B 0,C 180,E1 -17736.015,E2 -17736.015} C_VEL
LIN {X 0,Y 268.713,Z 550.006,A -85,B 0,C 180,E1 -17739.028,E2 -17739.028} C_VEL
LIN {X 0,Y 269.564,Z 545.104,A -85,B 0,C 180,E1 -17742.039,E2 -17742.039} C_VEL
LIN {X 0,Y 271.158,Z 538.566,A -85,B 0,C 180,E1 -17745.022,E2 -17745.022} C_VEL
LIN {X 0,Y 272.695,Z 531.578,A -85,B 0,C 180,E1 -17747.527,E2 -17747.527} C_VEL
LIN {X 0,Y 274.638,Z 523.662,A -85,B 0,C 180,E1 -17749.82,E2 -17749.82} C_VEL
LIN {X 0,Y 276.923,Z 514.514,A -85,B 0,C 180,E1 -17751.983,E2 -17751.983} C_VEL
LIN {X 0,Y 279.556,Z 503.416,A -85,B 0,C 180,E1 -17754.112,E2 -17754.112} C_VEL
LIN {X 0,Y 282.081,Z 492.149,A -85,B 0,C 180,E1 -17755.84,E2 -17755.84} C_VEL
LIN {X 0,Y 283.842,Z 482.601,A -85,B 0,C 180,E1 -17757.062,E2 -17757.062} C_VEL
LIN {X 0,Y 282.948,Z 471.819,A -85,B 0,C 180,E1 -17758.487,E2 -17758.487} C_VEL
LIN {X 0,Y 280.957,Z 460.301,A -85,B 0,C 180,E1 -17759.889,E2 -17759.889} C_VEL
LIN {X 0,Y 277.766,Z 446.691,A -85,B 0,C 180,E1 -17761.368,E2 -17761.368} C_VEL
LIN {X 0,Y 274.023,Z 435.104,A -85,B 0,C 180,E1 -17762.542,E2 -17762.542} C_VEL
LIN {X 0,Y 270.639,Z 425.833,A -85,B 0,C 180,E1 -17763.397,E2 -17763.397} C_VEL
LIN {X 0,Y 270.573,Z 425.23,A -85,B 0,C 180,E1 -17763.448,E2 -17763.448} C_VEL
LIN {X 0,Y 271.043,Z 421.992,A -85,B 0,C 180,E1 -17766.611,E2 -17766.611} C_VEL
LIN {X 0,Y 271.304,Z 419.662,A -85,B 0,C 180,E1 -17769.001,E2 -17769.001} C_VEL
LIN {X 0,Y 271.209,Z 416.544,A -85,B 0,C 180,E1 -17772.357,E2 -17772.357} C_VEL
LIN {X 0,Y 270.805,Z 412.921,A -85,B 0,C 180,E1 -17776.607,E2 -17776.607} C_VEL
LIN {X 0,Y 270.435,Z 410.638,A -85,B 0,C 180,E1 -17779.482,E2 -17779.482} C_VEL
LIN {X 0,Y 270.245,Z 409.449,A -85,B 0,C 180,E1 -17781.381,E2 -17781.381} C_VEL
LIN {X 0,Y 270.217,Z 409.453,A -85,B 0,C 180,E1 -17785.097,E2 -17785.097} C_VEL
LIN {X 0,Y 270.201,Z 409.456,A -85,B 0,C 180,E1 -17789.131,E2 -17789.131} C_VEL
LIN {X 0,Y 270.264,Z 409.447,A -85,B 0,C 180,E1 -17792.146,E2 -17792.146} C_VEL
LIN {X 0,Y 270.238,Z 409.449,A -85,B 0,C 180,E1 -17795.538,E2 -17795.538} C_VEL
LIN {X 0,Y 270.302,Z 409.441,A -85,B 0,C 180,E1 -17800.245,E2 -17800.245} C_VEL
LIN {X 0,Y 270.404,Z 409.426,A -85,B 0,C 180,E1 -17804.936,E2 -17804.936} C_VEL
LIN {X 0,Y 270.443,Z 409.419,A -85,B 0,C 180,E1 -17809.519,E2 -17809.519} C_VEL
LIN {X 0,Y 270.613,Z 409.395,A -85,B 0,C 180,E1 -17812.539,E2 -17812.539} C_VEL
LIN {X 0,Y 270.789,Z 409.381,A -85,B 0,C 180,E1 -17818.513,E2 -17818.513} C_VEL
LIN {X 0,Y 270.789,Z 409.381,A -85,B 0,C 180,E1 -17821.487,E2 -17821.487} C_VEL
LIN {X 0,Y 270.613,Z 409.401,A -85,B 0,C 180,E1 -17827.461,E2 -17827.461} C_VEL
LIN {X 0,Y 270.443,Z 409.421,A -85,B 0,C 180,E1 -17830.481,E2 -17830.481} C_VEL
LIN {X 0,Y 270.404,Z 409.428,A -85,B 0,C 180,E1 -17835.065,E2 -17835.065} C_VEL
LIN {X 0,Y 270.303,Z 409.441,A -85,B 0,C 180,E1 -17839.756,E2 -17839.756} C_VEL
LIN {X 0,Y 270.275,Z 409.444,A -85,B 0,C 180,E1 -17844.586,E2 -17844.586} C_VEL
LIN {X 0,Y 270.271,Z 409.445,A -85,B 0,C 180,E1 -17847.909,E2 -17847.909} C_VEL
LIN {X 0,Y 270.185,Z 409.455,A -85,B 0,C 180,E1 -17851.348,E2 -17851.348} C_VEL
LIN {X 0,Y 270.216,Z 409.451,A -85,B 0,C 180,E1 -17854.904,E2 -17854.904} C_VEL
LIN {X 0,Y 270.223,Z 409.45,A -85,B 0,C 180,E1 -17858.717,E2 -17858.717} C_VEL
LIN {X 0,Y 270.214,Z 409.606,A -85,B 0,C 180,E1 -17862.55,E2 -17862.55} C_VEL
LIN {X 0,Y 270.638,Z 412.656,A -85,B 0,C 180,E1 -17866.645,E2 -17866.645} C_VEL
LIN {X 0,Y 270.835,Z 414.988,A -85,B 0,C 180,E1 -17869.554,E2 -17869.554} C_VEL
LIN {X 0,Y 270.659,Z 418.212,A -85,B 0,C 180,E1 -17873.329,E2 -17873.329} C_VEL
LIN {X 0,Y 270.355,Z 421.205,A -85,B 0,C 180,E1 -17876.599,E2 -17876.599} C_VEL
LIN {X 0,Y 271.388,Z 424.384,A -85,B 0,C 180,E1 -17876.86,E2 -17876.86} C_VEL
LIN {X 0,Y 276.544,Z 437.904,A -85,B 0,C 180,E1 -17878.242,E2 -17878.242} C_VEL
LIN {X 0,Y 279.869,Z 449.349,A -85,B 0,C 180,E1 -17879.485,E2 -17879.485} C_VEL
LIN {X 0,Y 282.514,Z 461.376,A -85,B 0,C 180,E1 -17880.903,E2 -17880.903} C_VEL
LIN {X 0,Y 284.347,Z 473.212,A -85,B 0,C 180,E1 -17882.454,E2 -17882.454} C_VEL
LIN {X 0,Y 284.387,Z 476.823,A -85,B 0,C 180,E1 -17882.918,E2 -17882.918} C_VEL
LIN {X 0,Y 282.006,Z 489.309,A -85,B 0,C 180,E1 -17884.539,E2 -17884.539} C_VEL
LIN {X 0,Y 279.446,Z 500.21,A -85,B 0,C 180,E1 -17886.272,E2 -17886.272} C_VEL
LIN {X 0,Y 276.989,Z 510.964,A -85,B 0,C 180,E1 -17888.414,E2 -17888.414} C_VEL
LIN {X 0,Y 274.7,Z 519.84,A -85,B 0,C 180,E1 -17890.574,E2 -17890.574} C_VEL
LIN {X 0,Y 272.9,Z 527.224,A -85,B 0,C 180,E1 -17892.773,E2 -17892.773} C_VEL
LIN {X 0,Y 271.478,Z 533.375,A -85,B 0,C 180,E1 -17894.997,E2 -17894.997} C_VEL
LIN {X 0,Y 270.192,Z 538.462,A -85,B 0,C 180,E1 -17897.227,E2 -17897.227} C_VEL
LIN {X 0,Y 269.323,Z 542.541,A -85,B 0,C 180,E1 -17899.475,E2 -17899.475} C_VEL
LIN {X 0,Y 268.62,Z 546.672,A -85,B 0,C 180,E1 -17902.483,E2 -17902.483} C_VEL
LIN {X 0,Y 268.222,Z 549.373,A -85,B 0,C 180,E1 -17905.492,E2 -17905.492} C_VEL
LIN {X 0,Y 268.143,Z 550.723,A -85,B 0,C 180,E1 -17908.498,E2 -17908.498} C_VEL
LIN {X 0,Y 268.143,Z 550.752,A -85,B 0,C 180,E1 -17911.502,E2 -17911.502} C_VEL
LIN {X 0,Y 268.225,Z 549.456,A -85,B 0,C 180,E1 -17914.509,E2 -17914.509} C_VEL
LIN {X 0,Y 268.603,Z 546.806,A -85,B 0,C 180,E1 -17917.517,E2 -17917.517} C_VEL
LIN {X 0,Y 269.293,Z 542.732,A -85,B 0,C 180,E1 -17920.526,E2 -17920.526} C_VEL
LIN {X 0,Y 270.498,Z 537.105,A -85,B 0,C 180,E1 -17923.523,E2 -17923.523} C_VEL
LIN {X 0,Y 272.205,Z 530.748,A -85,B 0,C 180,E1 -17926.114,E2 -17926.114} C_VEL
LIN {X 0,Y 273.948,Z 523.094,A -85,B 0,C 180,E1 -17928.627,E2 -17928.627} C_VEL
LIN {X 0,Y 276.111,Z 514.58,A -85,B 0,C 180,E1 -17930.876,E2 -17930.876} C_VEL
LIN {X 0,Y 278.591,Z 504.617,A -85,B 0,C 180,E1 -17933.018,E2 -17933.018} C_VEL
LIN {X 0,Y 281.127,Z 493.525,A -85,B 0,C 180,E1 -17934.953,E2 -17934.953} C_VEL
LIN {X 0,Y 283.618,Z 481.325,A -85,B 0,C 180,E1 -17936.653,E2 -17936.653} C_VEL
LIN {X 0,Y 284.596,Z 475.53,A -85,B 0,C 180,E1 -17937.347,E2 -17937.347} C_VEL
LIN {X 0,Y 282.999,Z 463.889,A -85,B 0,C 180,E1 -17938.907,E2 -17938.907} C_VEL
LIN {X 0,Y 280.432,Z 451.496,A -85,B 0,C 180,E1 -17940.4,E2 -17940.4} C_VEL
LIN {X 0,Y 277.85,Z 442.133,A -85,B 0,C 180,E1 -17941.436,E2 -17941.436} C_VEL
LIN {X 0,Y 273.063,Z 428.257,A -85,B 0,C 180,E1 -17942.869,E2 -17942.869} C_VEL
LIN {X 0,Y 270.525,Z 422.149,A -85,B 0,C 180,E1 -17943.472,E2 -17943.472} C_VEL
LIN {X 0,Y 270.342,Z 421.123,A -85,B 0,C 180,E1 -17943.574,E2 -17943.574} C_VEL
LIN {X 0,Y 270.658,Z 418.331,A -85,B 0,C 180,E1 -17946.672,E2 -17946.672} C_VEL
LIN {X 0,Y 270.838,Z 415.078,A -85,B 0,C 180,E1 -17950.446,E2 -17950.446} C_VEL
LIN {X 0,Y 270.657,Z 412.76,A -85,B 0,C 180,E1 -17953.359,E2 -17953.359} C_VEL
LIN {X 0,Y 270.205,Z 409.722,A -85,B 0,C 180,E1 -17957.448,E2 -17957.448} C_VEL
LIN {X 0,Y 270.209,Z 409.453,A -85,B 0,C 180,E1 -17961.374,E2 -17961.374} C_VEL
LIN {X 0,Y 270.204,Z 409.453,A -85,B 0,C 180,E1 -17965.095,E2 -17965.095} C_VEL
LIN {X 0,Y 270.203,Z 409.454,A -85,B 0,C 180,E1 -17969.131,E2 -17969.131} C_VEL
LIN {X 0,Y 270.267,Z 409.446,A -85,B 0,C 180,E1 -17972.146,E2 -17972.146} C_VEL
LIN {X 0,Y 270.28,Z 409.442,A -85,B 0,C 180,E1 -17975.519,E2 -17975.519} C_VEL
LIN {X 0,Y 270.304,Z 409.435,A -85,B 0,C 180,E1 -17980.245,E2 -17980.245} C_VEL
LIN {X 0,Y 270.406,Z 409.426,A -85,B 0,C 180,E1 -17984.935,E2 -17984.935} C_VEL
LIN {X 0,Y 270.444,Z 409.422,A -85,B 0,C 180,E1 -17989.519,E2 -17989.519} C_VEL
LIN {X 0,Y 270.614,Z 409.401,A -85,B 0,C 180,E1 -17992.539,E2 -17992.539} C_VEL
LIN {X 0,Y 270.789,Z 409.379,A -85,B 0,C 180,E1 -17998.513,E2 -17998.513} C_VEL
LIN {X 0,Y 270.79,Z 409.379,A -85,B 0,C 180,E1 -18001.487,E2 -18001.487} C_VEL
LIN {X 0,Y 270.614,Z 409.401,A -85,B 0,C 180,E1 -18007.461,E2 -18007.461} C_VEL
LIN {X 0,Y 270.444,Z 409.421,A -85,B 0,C 180,E1 -18010.481,E2 -18010.481} C_VEL
LIN {X 0,Y 270.404,Z 409.427,A -85,B 0,C 180,E1 -18015.09,E2 -18015.09} C_VEL
LIN {X 0,Y 269.683,Z 409.518,A -85,B 0,C 180,E1 -18016.331,E2 -18016.331} C_VEL
LIN {X 0,Y 266.773,Z 409.88,A -85,B 0,C 180,E1 -18018.353,E2 -18018.353} C_VEL
LIN {X 0,Y 264.321,Z 410.186,A -85,B 0,C 180,E1 -18019.997,E2 -18019.997} C_VEL
LIN {X 0,Y 263.258,Z 410.317,A -85,B 0,C 180,E1 -18021.273,E2 -18021.273} C_VEL
LIN {X 0,Y 263.165,Z 410.328,A -85,B 0,C 180,E1 -18021.705,E2 -18021.705} C_VEL
LIN {X 0,Y 263.21,Z 410.323,A -85,B 0,C 180,E1 -18025.291,E2 -18025.291} C_VEL
LIN {X 0,Y 263.181,Z 410.328,A -85,B 0,C 180,E1 -18028.729,E2 -18028.729} C_VEL
LIN {X 0,Y 263.135,Z 410.335,A -85,B 0,C 180,E1 -18032.288,E2 -18032.288} C_VEL
LIN {X 0,Y 263.192,Z 410.33,A -85,B 0,C 180,E1 -18035.977,E2 -18035.977} C_VEL
LIN {X 0,Y 263.19,Z 410.331,A -85,B 0,C 180,E1 -18037.892,E2 -18037.892} C_VEL
LIN {X 0,Y 263.353,Z 411.48,A -85,B 0,C 180,E1 -18039.827,E2 -18039.827} C_VEL
LIN {X 0,Y 263.894,Z 414.698,A -85,B 0,C 180,E1 -18044.023,E2 -18044.023} C_VEL
LIN {X 0,Y 264.138,Z 416.531,A -85,B 0,C 180,E1 -18046.228,E2 -18046.228} C_VEL
LIN {X 0,Y 264.269,Z 418.337,A -85,B 0,C 180,E1 -18048.329,E2 -18048.329} C_VEL
LIN {X 0,Y 264.295,Z 420.253,A -85,B 0,C 180,E1 -18050.458,E2 -18050.458} C_VEL
LIN {X 0,Y 263.864,Z 423.785,A -85,B 0,C 180,E1 -18054.128,E2 -18054.128} C_VEL
LIN {X 0,Y 263.635,Z 425.159,A -85,B 0,C 180,E1 -18055.522,E2 -18055.522} C_VEL
LIN {X 0,Y 264.72,Z 428.563,A -85,B 0,C 180,E1 -18055.819,E2 -18055.819} C_VEL
LIN {X 0,Y 269.128,Z 440.509,A -85,B 0,C 180,E1 -18057.06,E2 -18057.06} C_VEL
LIN {X 0,Y 272.521,Z 451.995,A -85,B 0,C 180,E1 -18058.324,E2 -18058.324} C_VEL
LIN {X 0,Y 275.242,Z 465.062,A -85,B 0,C 180,E1 -18059.867,E2 -18059.867} C_VEL
LIN {X 0,Y 276.848,Z 476.699,A -85,B 0,C 180,E1 -18061.39,E2 -18061.39} C_VEL
LIN {X 0,Y 277.379,Z 483.301,A -85,B 0,C 180,E1 -18062.333,E2 -18062.333} C_VEL
LIN {X 0,Y 274.87,Z 495.922,A -85,B 0,C 180,E1 -18064.054,E2 -18064.054} C_VEL
LIN {X 0,Y 272.085,Z 507.427,A -85,B 0,C 180,E1 -18065.994,E2 -18065.994} C_VEL
LIN {X 0,Y 269.5,Z 517.827,A -85,B 0,C 180,E1 -18068.185,E2 -18068.185} C_VEL
LIN {X 0,Y 267.245,Z 526.408,A -85,B 0,C 180,E1 -18070.409,E2 -18070.409} C_VEL
LIN {X 0,Y 265.202,Z 534.622,A -85,B 0,C 180,E1 -18073.052,E2 -18073.052} C_VEL
LIN {X 0,Y 263.787,Z 540.377,A -85,B 0,C 180,E1 -18075.338,E2 -18075.338} C_VEL
LIN {X 0,Y 262.582,Z 545.088,A -85,B 0,C 180,E1 -18077.636,E2 -18077.636} C_VEL
LIN {X 0,Y 261.688,Z 549.973,A -85,B 0,C 180,E1 -18080.727,E2 -18080.727} C_VEL
LIN {X 0,Y 261.15,Z 553.368,A -85,B 0,C 180,E1 -18083.82,E2 -18083.82} C_VEL
LIN {X 0,Y 261.007,Z 555.375,A -85,B 0,C 180,E1 -18086.913,E2 -18086.913} C_VEL
LIN {X 0,Y 261.072,Z 556.037,A -85,B 0,C 180,E1 -18090,E2 -18090} C_VEL
LIN {X 0,Y 261.007,Z 555.363,A -85,B 0,C 180,E1 -18093.087,E2 -18093.087} C_VEL
LIN {X 0,Y 261.163,Z 553.346,A -85,B 0,C 180,E1 -18096.179,E2 -18096.179} C_VEL
LIN {X 0,Y 261.685,Z 549.937,A -85,B 0,C 180,E1 -18099.273,E2 -18099.273} C_VEL
LIN {X 0,Y 262.579,Z 545.033,A -85,B 0,C 180,E1 -18102.364,E2 -18102.364} C_VEL
LIN {X 0,Y 264.244,Z 538.495,A -85,B 0,C 180,E1 -18105.424,E2 -18105.424} C_VEL
LIN {X 0,Y 265.768,Z 531.992,A -85,B 0,C 180,E1 -18107.826,E2 -18107.826} C_VEL
LIN {X 0,Y 267.923,Z 523.591,A -85,B 0,C 180,E1 -18110.338,E2 -18110.338} C_VEL
LIN {X 0,Y 270.335,Z 514.442,A -85,B 0,C 180,E1 -18112.548,E2 -18112.548} C_VEL
LIN {X 0,Y 272.57,Z 505.32,A -85,B 0,C 180,E1 -18114.365,E2 -18114.365} C_VEL
LIN {X 0,Y 275.329,Z 493.574,A -85,B 0,C 180,E1 -18116.274,E2 -18116.274} C_VEL
LIN {X 0,Y 277.258,Z 483.954,A -85,B 0,C 180,E1 -18117.554,E2 -18117.554} C_VEL
LIN {X 0,Y 276.629,Z 474.614,A -85,B 0,C 180,E1 -18118.863,E2 -18118.863} C_VEL
LIN {X 0,Y 274.603,Z 461.775,A -85,B 0,C 180,E1 -18120.508,E2 -18120.508} C_VEL
LIN {X 0,Y 271.548,Z 448.623,A -85,B 0,C 180,E1 -18122.027,E2 -18122.027} C_VEL
LIN {X 0,Y 267.554,Z 435.877,A -85,B 0,C 180,E1 -18123.388,E2 -18123.388} C_VEL
LIN {X 0,Y 264.625,Z 428.391,A -85,B 0,C 180,E1 -18124.159,E2 -18124.159} C_VEL
LIN {X 0,Y 263.629,Z 425.123,A -85,B 0,C 180,E1 -18124.476,E2 -18124.476} C_VEL
LIN {X 0,Y 264.117,Z 421.932,A -85,B 0,C 180,E1 -18127.735,E2 -18127.735} C_VEL
LIN {X 0,Y 264.292,Z 420.111,A -85,B 0,C 180,E1 -18129.658,E2 -18129.658} C_VEL
LIN {X 0,Y 264.234,Z 418.129,A -85,B 0,C 180,E1 -18131.864,E2 -18131.864} C_VEL
LIN {X 0,Y 263.877,Z 414.657,A -85,B 0,C 180,E1 -18135.981,E2 -18135.981} C_VEL
LIN {X 0,Y 263.341,Z 411.431,A -85,B 0,C 180,E1 -18140.17,E2 -18140.17} C_VEL
LIN {X 0,Y 263.189,Z 410.327,A -85,B 0,C 180,E1 -18142.108,E2 -18142.108} C_VEL
LIN {X 0,Y 263.184,Z 410.329,A -85,B 0,C 180,E1 -18145.89,E2 -18145.89} C_VEL
LIN {X 0,Y 263.141,Z 410.335,A -85,B 0,C 180,E1 -18149.506,E2 -18149.506} C_VEL
LIN {X 0,Y 263.191,Z 410.327,A -85,B 0,C 180,E1 -18153.003,E2 -18153.003} C_VEL
LIN {X 0,Y 263.156,Z 410.331,A -85,B 0,C 180,E1 -18156.384,E2 -18156.384} C_VEL
LIN {X 0,Y 263.264,Z 410.316,A -85,B 0,C 180,E1 -18159.693,E2 -18159.693} C_VEL
LIN {X 0,Y 263.352,Z 410.305,A -85,B 0,C 180,E1 -18164.522,E2 -18164.522} C_VEL
LIN {X 0,Y 263.375,Z 410.298,A -85,B 0,C 180,E1 -18169.235,E2 -18169.235} C_VEL
LIN {X 0,Y 263.574,Z 410.273,A -85,B 0,C 180,E1 -18172.339,E2 -18172.339} C_VEL
LIN {X 0,Y 263.753,Z 410.257,A -85,B 0,C 180,E1 -18178.473,E2 -18178.473} C_VEL
LIN {X 0,Y 263.753,Z 410.257,A -85,B 0,C 180,E1 -18181.527,E2 -18181.527} C_VEL
LIN {X 0,Y 263.574,Z 410.279,A -85,B 0,C 180,E1 -18187.662,E2 -18187.662} C_VEL
LIN {X 0,Y 263.375,Z 410.302,A -85,B 0,C 180,E1 -18190.766,E2 -18190.766} C_VEL
LIN {X 0,Y 263.352,Z 410.306,A -85,B 0,C 180,E1 -18195.478,E2 -18195.478} C_VEL
LIN {X 0,Y 263.265,Z 410.317,A -85,B 0,C 180,E1 -18200.307,E2 -18200.307} C_VEL
LIN {X 0,Y 263.21,Z 410.324,A -85,B 0,C 180,E1 -18205.291,E2 -18205.291} C_VEL
LIN {X 0,Y 263.167,Z 410.329,A -85,B 0,C 180,E1 -18208.731,E2 -18208.731} C_VEL
LIN {X 0,Y 263.134,Z 410.334,A -85,B 0,C 180,E1 -18212.288,E2 -18212.288} C_VEL
LIN {X 0,Y 263.189,Z 410.328,A -85,B 0,C 180,E1 -18215.978,E2 -18215.978} C_VEL
LIN {X 0,Y 263.116,Z 410.335,A -85,B 0,C 180,E1 -18219.871,E2 -18219.871} C_VEL
LIN {X 0,Y 263.142,Z 410.409,A -85,B 0,C 180,E1 -18221.89,E2 -18221.89} C_VEL
LIN {X 0,Y 263.561,Z 413.427,A -85,B 0,C 180,E1 -18226.108,E2 -18226.108} C_VEL
LIN {X 0,Y 263.761,Z 415.066,A -85,B 0,C 180,E1 -18228.251,E2 -18228.251} C_VEL
LIN {X 0,Y 263.797,Z 416.953,A -85,B 0,C 180,E1 -18230.589,E2 -18230.589} C_VEL
LIN {X 0,Y 263.544,Z 419.903,A -85,B 0,C 180,E1 -18234.078,E2 -18234.078} C_VEL
LIN {X 0,Y 263.394,Z 421.216,A -85,B 0,C 180,E1 -18235.569,E2 -18235.569} C_VEL
LIN {X 0,Y 264.402,Z 424.381,A -85,B 0,C 180,E1 -18235.862,E2 -18235.862} C_VEL
LIN {X 0,Y 267.866,Z 432.79,A -85,B 0,C 180,E1 -18236.765,E2 -18236.765} C_VEL
LIN {X 0,Y 271.936,Z 444.869,A -85,B 0,C 180,E1 -18238.121,E2 -18238.121} C_VEL
LIN {X 0,Y 275.022,Z 457.238,A -85,B 0,C 180,E1 -18239.594,E2 -18239.594} C_VEL
LIN {X 0,Y 277.173,Z 469.524,A -85,B 0,C 180,E1 -18241.199,E2 -18241.199} C_VEL
LIN {X 0,Y 278.052,Z 476.613,A -85,B 0,C 180,E1 -18242.209,E2 -18242.209} C_VEL
LIN {X 0,Y 275.868,Z 488.205,A -85,B 0,C 180,E1 -18243.727,E2 -18243.727} C_VEL
LIN {X 0,Y 273.528,Z 498.291,A -85,B 0,C 180,E1 -18245.322,E2 -18245.322} C_VEL
LIN {X 0,Y 271.168,Z 507.704,A -85,B 0,C 180,E1 -18247.123,E2 -18247.123} C_VEL
LIN {X 0,Y 268.726,Z 517.163,A -85,B 0,C 180,E1 -18249.325,E2 -18249.325} C_VEL
LIN {X 0,Y 266.533,Z 525.358,A -85,B 0,C 180,E1 -18251.67,E2 -18251.67} C_VEL
LIN {X 0,Y 265.163,Z 531.515,A -85,B 0,C 180,E1 -18253.842,E2 -18253.842} C_VEL
LIN {X 0,Y 263.604,Z 536.926,A -85,B 0,C 180,E1 -18256.116,E2 -18256.116} C_VEL
LIN {X 0,Y 262.33,Z 542.611,A -85,B 0,C 180,E1 -18259.191,E2 -18259.191} C_VEL
LIN {X 0,Y 261.559,Z 546.742,A -85,B 0,C 180,E1 -18262.279,E2 -18262.279} C_VEL
LIN {X 0,Y 261.144,Z 549.442,A -85,B 0,C 180,E1 -18265.369,E2 -18265.369} C_VEL
LIN {X 0,Y 261.052,Z 550.792,A -85,B 0,C 180,E1 -18268.457,E2 -18268.457} C_VEL
LIN {X 0,Y 261.075,Z 550.971,A -85,B 0,C 180,E1 -18270,E2 -18270} C_VEL
LIN {X 0,Y 261.081,Z 550.339,A -85,B 0,C 180,E1 -18273.086,E2 -18273.086} C_VEL
LIN {X 0,Y 261.321,Z 548.371,A -85,B 0,C 180,E1 -18276.176,E2 -18276.176} C_VEL
LIN {X 0,Y 261.862,Z 545.022,A -85,B 0,C 180,E1 -18279.267,E2 -18279.267} C_VEL
LIN {X 0,Y 262.898,Z 540.19,A -85,B 0,C 180,E1 -18282.349,E2 -18282.349} C_VEL
LIN {X 0,Y 264.072,Z 535.526,A -85,B 0,C 180,E1 -18284.645,E2 -18284.645} C_VEL
LIN {X 0,Y 265.544,Z 529.811,A -85,B 0,C 180,E1 -18286.926,E2 -18286.926} C_VEL
LIN {X 0,Y 267.609,Z 521.669,A -85,B 0,C 180,E1 -18289.563,E2 -18289.563} C_VEL
LIN {X 0,Y 269.88,Z 513.148,A -85,B 0,C 180,E1 -18291.783,E2 -18291.783} C_VEL
LIN {X 0,Y 272.492,Z 502.817,A -85,B 0,C 180,E1 -18293.968,E2 -18293.968} C_VEL
LIN {X 0,Y 275.248,Z 491.259,A -85,B 0,C 180,E1 -18295.929,E2 -18295.929} C_VEL
LIN {X 0,Y 277.779,Z 478.579,A -85,B 0,C 180,E1 -18297.662,E2 -18297.662} C_VEL
LIN {X 0,Y 277.829,Z 474.69,A -85,B 0,C 180,E1 -18298.19,E2 -18298.19} C_VEL
LIN {X 0,Y 276.341,Z 464.002,A -85,B 0,C 180,E1 -18299.668,E2 -18299.668} C_VEL
LIN {X 0,Y 273.654,Z 451.058,A -85,B 0,C 180,E1 -18301.278,E2 -18301.278} C_VEL
LIN {X 0,Y 269.747,Z 438.107,A -85,B 0,C 180,E1 -18302.779,E2 -18302.779} C_VEL
LIN {X 0,Y 264.909,Z 425.137,A -85,B 0,C 180,E1 -18304.167,E2 -18304.167} C_VEL
LIN {X 0,Y 263.545,Z 422.038,A -85,B 0,C 180,E1 -18304.488,E2 -18304.488} C_VEL
LIN {X 0,Y 263.43,Z 421.197,A -85,B 0,C 180,E1 -18304.582,E2 -18304.582} C_VEL
LIN {X 0,Y 263.694,Z 418.385,A -85,B 0,C 180,E1 -18307.807,E2 -18307.807} C_VEL
LIN {X 0,Y 263.806,Z 416.771,A -85,B 0,C 180,E1 -18309.746,E2 -18309.746} C_VEL
LIN {X 0,Y 263.756,Z 415.162,A -85,B 0,C 180,E1 -18311.771,E2 -18311.771} C_VEL
LIN {X 0,Y 263.582,Z 413.493,A -85,B 0,C 180,E1 -18313.952,E2 -18313.952} C_VEL
LIN {X 0,Y 263.139,Z 410.525,A -85,B 0,C 180,E1 -18318.109,E2 -18318.109} C_VEL
LIN {X 0,Y 263.161,Z 410.329,A -85,B 0,C 180,E1 -18322.103,E2 -18322.103} C_VEL
LIN {X 0,Y 263.153,Z 410.33,A -85,B 0,C 180,E1 -18325.886,E2 -18325.886} C_VEL
LIN {X 0,Y 263.153,Z 410.331,A -85,B 0,C 180,E1 -18329.507,E2 -18329.507} C_VEL
LIN {X 0,Y 263.195,Z 410.326,A -85,B 0,C 180,E1 -18333.003,E2 -18333.003} C_VEL
LIN {X 0,Y 263.187,Z 410.322,A -85,B 0,C 180,E1 -18336.387,E2 -18336.387} C_VEL
LIN {X 0,Y 263.266,Z 410.31,A -85,B 0,C 180,E1 -18339.693,E2 -18339.693} C_VEL
LIN {X 0,Y 263.354,Z 410.304,A -85,B 0,C 180,E1 -18344.522,E2 -18344.522} C_VEL
LIN {X 0,Y 263.377,Z 410.303,A -85,B 0,C 180,E1 -18349.234,E2 -18349.234} C_VEL
LIN {X 0,Y 263.576,Z 410.279,A -85,B 0,C 180,E1 -18352.338,E2 -18352.338} C_VEL
LIN {X 0,Y 263.753,Z 410.255,A -85,B 0,C 180,E1 -18358.473,E2 -18358.473} C_VEL
LIN {X 0,Y 263.755,Z 410.255,A -85,B 0,C 180,E1 -18361.527,E2 -18361.527} C_VEL
LIN {X 0,Y 263.576,Z 410.278,A -85,B 0,C 180,E1 -18367.661,E2 -18367.661} C_VEL
LIN {X 0,Y 263.377,Z 410.302,A -85,B 0,C 180,E1 -18370.765,E2 -18370.765} C_VEL
LIN {X 0,Y 263.353,Z 410.306,A -85,B 0,C 180,E1 -18375.478,E2 -18375.478} C_VEL
LIN {X 0,Y 263.266,Z 410.317,A -85,B 0,C 180,E1 -18380.306,E2 -18380.306} C_VEL
LIN {X 0,Y 263.165,Z 410.328,A -85,B 0,C 180,E1 -18381.705,E2 -18381.705} C_VEL
LIN {X 0,Y 262.477,Z 410.417,A -85,B 0,C 180,E1 -18382.983,E2 -18382.983} C_VEL
LIN {X 0,Y 259.619,Z 410.77,A -85,B 0,C 180,E1 -18385.067,E2 -18385.067} C_VEL
LIN {X 0,Y 257.219,Z 411.066,A -85,B 0,C 180,E1 -18386.761,E2 -18386.761} C_VEL
LIN {X 0,Y 256.21,Z 411.194,A -85,B 0,C 180,E1 -18388.075,E2 -18388.075} C_VEL
LIN {X 0,Y 256.138,Z 411.204,A -85,B 0,C 180,E1 -18388.52,E2 -18388.52} C_VEL
LIN {X 0,Y 256.087,Z 411.213,A -85,B 0,C 180,E1 -18393.29,E2 -18393.29} C_VEL
LIN {X 0,Y 256.143,Z 411.209,A -85,B 0,C 180,E1 -18397.279,E2 -18397.279} C_VEL
LIN {X 0,Y 256.498,Z 413.733,A -85,B 0,C 180,E1 -18401.117,E2 -18401.117} C_VEL
LIN {X 0,Y 257.023,Z 416.95,A -85,B 0,C 180,E1 -18405.312,E2 -18405.312} C_VEL
LIN {X 0,Y 257.22,Z 418.799,A -85,B 0,C 180,E1 -18407.537,E2 -18407.537} C_VEL
LIN {X 0,Y 257.198,Z 421.884,A -85,B 0,C 180,E1 -18411.062,E2 -18411.062} C_VEL
LIN {X 0,Y 256.765,Z 425.107,A -85,B 0,C 180,E1 -18414.469,E2 -18414.469} C_VEL
LIN {X 0,Y 257.787,Z 428.367,A -85,B 0,C 180,E1 -18414.761,E2 -18414.761} C_VEL
LIN {X 0,Y 262.303,Z 440.212,A -85,B 0,C 180,E1 -18416.074,E2 -18416.074} C_VEL
LIN {X 0,Y 266.26,Z 453.626,A -85,B 0,C 180,E1 -18417.634,E2 -18417.634} C_VEL
LIN {X 0,Y 268.779,Z 466.068,A -85,B 0,C 180,E1 -18419.181,E2 -18419.181} C_VEL
LIN {X 0,Y 270.358,Z 478.059,A -85,B 0,C 180,E1 -18420.829,E2 -18420.829} C_VEL
LIN {X 0,Y 270.841,Z 484.106,A -85,B 0,C 180,E1 -18421.734,E2 -18421.734} C_VEL
LIN {X 0,Y 268.69,Z 494.989,A -85,B 0,C 180,E1 -18423.256,E2 -18423.256} C_VEL
LIN {X 0,Y 266.102,Z 505.408,A -85,B 0,C 180,E1 -18425.003,E2 -18425.003} C_VEL
LIN {X 0,Y 263.292,Z 516.131,A -85,B 0,C 180,E1 -18427.229,E2 -18427.229} C_VEL
LIN {X 0,Y 260.868,Z 524.984,A -85,B 0,C 180,E1 -18429.498,E2 -18429.498} C_VEL
LIN {X 0,Y 258.664,Z 532.87,A -85,B 0,C 180,E1 -18431.982,E2 -18431.982} C_VEL
LIN {X 0,Y 256.888,Z 540.309,A -85,B 0,C 180,E1 -18434.935,E2 -18434.935} C_VEL
LIN {X 0,Y 255.611,Z 545.02,A -85,B 0,C 180,E1 -18437.293,E2 -18437.293} C_VEL
LIN {X 0,Y 254.639,Z 549.904,A -85,B 0,C 180,E1 -18440.468,E2 -18440.468} C_VEL
LIN {X 0,Y 254.063,Z 553.299,A -85,B 0,C 180,E1 -18443.647,E2 -18443.647} C_VEL
LIN {X 0,Y 253.912,Z 555.307,A -85,B 0,C 180,E1 -18446.826,E2 -18446.826} C_VEL
LIN {X 0,Y 253.98,Z 555.968,A -85,B 0,C 180,E1 -18450,E2 -18450} C_VEL
LIN {X 0,Y 253.912,Z 555.294,A -85,B 0,C 180,E1 -18453.173,E2 -18453.173} C_VEL
LIN {X 0,Y 254.075,Z 553.276,A -85,B 0,C 180,E1 -18456.352,E2 -18456.352} C_VEL
LIN {X 0,Y 254.635,Z 549.867,A -85,B 0,C 180,E1 -18459.532,E2 -18459.532} C_VEL
LIN {X 0,Y 255.608,Z 544.963,A -85,B 0,C 180,E1 -18462.707,E2 -18462.707} C_VEL
LIN {X 0,Y 257.337,Z 538.424,A -85,B 0,C 180,E1 -18465.849,E2 -18465.849} C_VEL
LIN {X 0,Y 259.052,Z 531.682,A -85,B 0,C 180,E1 -18468.393,E2 -18468.393} C_VEL
LIN {X 0,Y 261.248,Z 523.519,A -85,B 0,C 180,E1 -18470.882,E2 -18470.882} C_VEL
LIN {X 0,Y 263.771,Z 514.371,A -85,B 0,C 180,E1 -18473.141,E2 -18473.141} C_VEL
LIN {X 0,Y 266.115,Z 505.248,A -85,B 0,C 180,E1 -18474.996,E2 -18474.996} C_VEL
LIN {X 0,Y 268.684,Z 494.755,A -85,B 0,C 180,E1 -18476.752,E2 -18476.752} C_VEL
LIN {X 0,Y 270.787,Z 483.873,A -85,B 0,C 180,E1 -18478.272,E2 -18478.272} C_VEL
LIN {X 0,Y 269.774,Z 472.97,A -85,B 0,C 180,E1 -18479.858,E2 -18479.858} C_VEL
LIN {X 0,Y 268.023,Z 462.14,A -85,B 0,C 180,E1 -18481.297,E2 -18481.297} C_VEL
LIN {X 0,Y 265.104,Z 449.574,A -85,B 0,C 180,E1 -18482.825,E2 -18482.825} C_VEL
LIN {X 0,Y 260.943,Z 436.309,A -85,B 0,C 180,E1 -18484.323,E2 -18484.323} C_VEL
LIN {X 0,Y 257.499,Z 427.799,A -85,B 0,C 180,E1 -18485.262,E2 -18485.262} C_VEL
LIN {X 0,Y 256.752,Z 425.061,A -85,B 0,C 180,E1 -18485.531,E2 -18485.531} C_VEL
LIN {X 0,Y 257.196,Z 421.846,A -85,B 0,C 180,E1 -18488.938,E2 -18488.938} C_VEL
LIN {X 0,Y 257.181,Z 418.773,A -85,B 0,C 180,E1 -18492.453,E2 -18492.453} C_VEL
LIN {X 0,Y 256.931,Z 416.395,A -85,B 0,C 180,E1 -18495.332,E2 -18495.332} C_VEL
LIN {X 0,Y 256.493,Z 413.687,A -85,B 0,C 180,E1 -18498.882,E2 -18498.882} C_VEL
LIN {X 0,Y 256.279,Z 412.219,A -85,B 0,C 180,E1 -18500.896,E2 -18500.896} C_VEL
LIN {X 0,Y 256.156,Z 411.204,A -85,B 0,C 180,E1 -18502.872,E2 -18502.872} C_VEL
LIN {X 0,Y 256.086,Z 411.214,A -85,B 0,C 180,E1 -18506.71,E2 -18506.71} C_VEL
LIN {X 0,Y 256.127,Z 411.207,A -85,B 0,C 180,E1 -18511.41,E2 -18511.41} C_VEL
LIN {X 0,Y 256.143,Z 411.205,A -85,B 0,C 180,E1 -18515.697,E2 -18515.697} C_VEL
LIN {X 0,Y 256.164,Z 411.203,A -85,B 0,C 180,E1 -18519.105,E2 -18519.105} C_VEL
LIN {X 0,Y 256.301,Z 411.185,A -85,B 0,C 180,E1 -18524.085,E2 -18524.085} C_VEL
LIN {X 0,Y 256.311,Z 411.178,A -85,B 0,C 180,E1 -18528.934,E2 -18528.934} C_VEL
LIN {X 0,Y 256.542,Z 411.15,A -85,B 0,C 180,E1 -18532.127,E2 -18532.127} C_VEL
LIN {X 0,Y 256.716,Z 411.133,A -85,B 0,C 180,E1 -18538.431,E2 -18538.431} C_VEL
LIN {X 0,Y 256.716,Z 411.133,A -85,B 0,C 180,E1 -18541.569,E2 -18541.569} C_VEL
LIN {X 0,Y 256.542,Z 411.156,A -85,B 0,C 180,E1 -18547.873,E2 -18547.873} C_VEL
LIN {X 0,Y 256.311,Z 411.182,A -85,B 0,C 180,E1 -18551.066,E2 -18551.066} C_VEL
LIN {X 0,Y 256.302,Z 411.185,A -85,B 0,C 180,E1 -18555.915,E2 -18555.915} C_VEL
LIN {X 0,Y 256.168,Z 411.202,A -85,B 0,C 180,E1 -18560.895,E2 -18560.895} C_VEL
LIN {X 0,Y 256.19,Z 411.198,A -85,B 0,C 180,E1 -18565.139,E2 -18565.139} C_VEL
LIN {X 0,Y 256.105,Z 411.209,A -85,B 0,C 180,E1 -18569.601,E2 -18569.601} C_VEL
LIN {X 0,Y 256.086,Z 411.212,A -85,B 0,C 180,E1 -18573.29,E2 -18573.29} C_VEL
LIN {X 0,Y 256.13,Z 411.207,A -85,B 0,C 180,E1 -18577.275,E2 -18577.275} C_VEL
LIN {X 0,Y 256.067,Z 411.229,A -85,B 0,C 180,E1 -18581.201,E2 -18581.201} C_VEL
LIN {X 0,Y 256.488,Z 414.143,A -85,B 0,C 180,E1 -18585.433,E2 -18585.433} C_VEL
LIN {X 0,Y 256.741,Z 416.735,A -85,B 0,C 180,E1 -18588.931,E2 -18588.931} C_VEL
LIN {X 0,Y 256.634,Z 419.681,A -85,B 0,C 180,E1 -18592.578,E2 -18592.578} C_VEL
LIN {X 0,Y 256.488,Z 421.375,A -85,B 0,C 180,E1 -18594.53,E2 -18594.53} C_VEL
LIN {X 0,Y 257.605,Z 424.641,A -85,B 0,C 180,E1 -18594.837,E2 -18594.837} C_VEL
LIN {X 0,Y 262.189,Z 435.956,A -85,B 0,C 180,E1 -18596.144,E2 -18596.144} C_VEL
LIN {X 0,Y 266.221,Z 448.482,A -85,B 0,C 180,E1 -18597.648,E2 -18597.648} C_VEL
LIN {X 0,Y 268.754,Z 459.121,A -85,B 0,C 180,E1 -18598.99,E2 -18598.99} C_VEL
LIN {X 0,Y 270.779,Z 471.246,A -85,B 0,C 180,E1 -18600.659,E2 -18600.659} C_VEL
LIN {X 0,Y 271.51,Z 477.877,A -85,B 0,C 180,E1 -18601.653,E2 -18601.653} C_VEL
LIN {X 0,Y 269.25,Z 489.455,A -85,B 0,C 180,E1 -18603.24,E2 -18603.24} C_VEL
LIN {X 0,Y 266.501,Z 500.355,A -85,B 0,C 180,E1 -18605.043,E2 -18605.043} C_VEL
LIN {X 0,Y 263.758,Z 511.108,A -85,B 0,C 180,E1 -18607.272,E2 -18607.272} C_VEL
LIN {X 0,Y 261.282,Z 519.983,A -85,B 0,C 180,E1 -18609.533,E2 -18609.533} C_VEL
LIN {X 0,Y 259.07,Z 528.252,A -85,B 0,C 180,E1 -18612.147,E2 -18612.147} C_VEL
LIN {X 0,Y 257.758,Z 533.517,A -85,B 0,C 180,E1 -18614.178,E2 -18614.178} C_VEL
LIN {X 0,Y 256.282,Z 538.603,A -85,B 0,C 180,E1 -18616.521,E2 -18616.521} C_VEL
LIN {X 0,Y 255.069,Z 543.872,A -85,B 0,C 180,E1 -18619.683,E2 -18619.683} C_VEL
LIN {X 0,Y 254.504,Z 546.812,A -85,B 0,C 180,E1 -18622.064,E2 -18622.064} C_VEL
LIN {X 0,Y 254.063,Z 549.511,A -85,B 0,C 180,E1 -18625.24,E2 -18625.24} C_VEL
LIN {X 0,Y 253.963,Z 550.861,A -85,B 0,C 180,E1 -18628.414,E2 -18628.414} C_VEL
LIN {X 0,Y 253.983,Z 551.04,A -85,B 0,C 180,E1 -18630,E2 -18630} C_VEL
LIN {X 0,Y 253.983,Z 550.408,A -85,B 0,C 180,E1 -18633.173,E2 -18633.173} C_VEL
LIN {X 0,Y 254.25,Z 548.44,A -85,B 0,C 180,E1 -18636.348,E2 -18636.348} C_VEL
LIN {X 0,Y 254.826,Z 545.09,A -85,B 0,C 180,E1 -18639.525,E2 -18639.525} C_VEL
LIN {X 0,Y 255.915,Z 540.259,A -85,B 0,C 180,E1 -18642.691,E2 -18642.691} C_VEL
LIN {X 0,Y 257.197,Z 535.594,A -85,B 0,C 180,E1 -18645.046,E2 -18645.046} C_VEL
LIN {X 0,Y 259.063,Z 528.603,A -85,B 0,C 180,E1 -18647.847,E2 -18647.847} C_VEL
LIN {X 0,Y 260.883,Z 521.737,A -85,B 0,C 180,E1 -18650.089,E2 -18650.089} C_VEL
LIN {X 0,Y 263.277,Z 513.214,A -85,B 0,C 180,E1 -18652.358,E2 -18652.358} C_VEL
LIN {X 0,Y 265.997,Z 502.883,A -85,B 0,C 180,E1 -18654.591,E2 -18654.591} C_VEL
LIN {X 0,Y 268.881,Z 491.324,A -85,B 0,C 180,E1 -18656.591,E2 -18656.591} C_VEL
LIN {X 0,Y 271.426,Z 479.005,A -85,B 0,C 180,E1 -18658.314,E2 -18658.314} C_VEL
LIN {X 0,Y 270.717,Z 470.633,A -85,B 0,C 180,E1 -18659.555,E2 -18659.555} C_VEL
LIN {X 0,Y 268.744,Z 459.103,A -85,B 0,C 180,E1 -18661.143,E2 -18661.143} C_VEL
LIN {X 0,Y 266.389,Z 449.073,A -85,B 0,C 180,E1 -18662.409,E2 -18662.409} C_VEL
LIN {X 0,Y 261.887,Z 435.017,A -85,B 0,C 180,E1 -18664.094,E2 -18664.094} C_VEL
LIN {X 0,Y 257.505,Z 424.422,A -85,B 0,C 180,E1 -18665.323,E2 -18665.323} C_VEL
LIN {X 0,Y 256.5,Z 421.287,A -85,B 0,C 180,E1 -18665.625,E2 -18665.625} C_VEL
LIN {X 0,Y 256.785,Z 417.708,A -85,B 0,C 180,E1 -18669.973,E2 -18669.973} C_VEL
LIN {X 0,Y 256.601,Z 415.23,A -85,B 0,C 180,E1 -18673.214,E2 -18673.214} C_VEL
LIN {X 0,Y 256.279,Z 412.741,A -85,B 0,C 180,E1 -18676.718,E2 -18676.718} C_VEL
LIN {X 0,Y 256.089,Z 411.332,A -85,B 0,C 180,E1 -18678.803,E2 -18678.803} C_VEL
LIN {X 0,Y 256.133,Z 411.207,A -85,B 0,C 180,E1 -18682.868,E2 -18682.868} C_VEL
LIN {X 0,Y 256.07,Z 411.214,A -85,B 0,C 180,E1 -18686.707,E2 -18686.707} C_VEL
LIN {X 0,Y 256.116,Z 411.205,A -85,B 0,C 180,E1 -18690.4,E2 -18690.4} C_VEL
LIN {X 0,Y 256.191,Z 411.198,A -85,B 0,C 180,E1 -18694.861,E2 -18694.861} C_VEL
LIN {X 0,Y 256.17,Z 411.196,A -85,B 0,C 180,E1 -18699.105,E2 -18699.105} C_VEL
LIN {X 0,Y 256.303,Z 411.183,A -85,B 0,C 180,E1 -18704.085,E2 -18704.085} C_VEL
LIN {X 0,Y 256.313,Z 411.182,A -85,B 0,C 180,E1 -18708.934,E2 -18708.934} C_VEL
LIN {X 0,Y 256.543,Z 411.156,A -85,B 0,C 180,E1 -18712.127,E2 -18712.127} C_VEL
LIN {X 0,Y 256.716,Z 411.132,A -85,B 0,C 180,E1 -18718.431,E2 -18718.431} C_VEL
LIN {X 0,Y 256.718,Z 411.132,A -85,B 0,C 180,E1 -18721.569,E2 -18721.569} C_VEL
LIN {X 0,Y 256.543,Z 411.154,A -85,B 0,C 180,E1 -18727.873,E2 -18727.873} C_VEL
LIN {X 0,Y 256.312,Z 411.183,A -85,B 0,C 180,E1 -18731.066,E2 -18731.066} C_VEL
LIN {X 0,Y 256.302,Z 411.185,A -85,B 0,C 180,E1 -18735.915,E2 -18735.915} C_VEL
LIN {X 0,Y 256.169,Z 411.201,A -85,B 0,C 180,E1 -18740.895,E2 -18740.895} C_VEL
LIN {X 0,Y 256.19,Z 411.197,A -85,B 0,C 180,E1 -18745.138,E2 -18745.138} C_VEL
LIN {X 0,Y 256.138,Z 411.204,A -85,B 0,C 180,E1 -18748.52,E2 -18748.52} C_VEL
LIN {X 0,Y 255.494,Z 411.292,A -85,B 0,C 180,E1 -18749.831,E2 -18749.831} C_VEL
LIN {X 0,Y 252.644,Z 411.65,A -85,B 0,C 180,E1 -18751.968,E2 -18751.968} C_VEL
LIN {X 0,Y 250.204,Z 411.949,A -85,B 0,C 180,E1 -18753.707,E2 -18753.707} C_VEL
LIN {X 0,Y 249.151,Z 412.078,A -85,B 0,C 180,E1 -18755.056,E2 -18755.056} C_VEL
LIN {X 0,Y 249.063,Z 412.088,A -85,B 0,C 180,E1 -18755.514,E2 -18755.514} C_VEL
LIN {X 0,Y 249.077,Z 412.089,A -85,B 0,C 180,E1 -18756.337,E2 -18756.337} C_VEL
LIN {X 0,Y 249.219,Z 413.079,A -85,B 0,C 180,E1 -18758.345,E2 -18758.345} C_VEL
LIN {X 0,Y 249.698,Z 416.014,A -85,B 0,C 180,E1 -18762.493,E2 -18762.493} C_VEL
LIN {X 0,Y 250.031,Z 418.188,A -85,B 0,C 180,E1 -18765.355,E2 -18765.355} C_VEL
LIN {X 0,Y 250.216,Z 420.001,A -85,B 0,C 180,E1 -18767.615,E2 -18767.615} C_VEL
LIN {X 0,Y 250.224,Z 421.823,A -85,B 0,C 180,E1 -18769.759,E2 -18769.759} C_VEL
LIN {X 0,Y 249.922,Z 425.099,A -85,B 0,C 180,E1 -18773.343,E2 -18773.343} C_VEL
LIN {X 0,Y 251.005,Z 428.417,A -85,B 0,C 180,E1 -18773.664,E2 -18773.664} C_VEL
LIN {X 0,Y 256.026,Z 441.428,A -85,B 0,C 180,E1 -18775.207,E2 -18775.207} C_VEL
LIN {X 0,Y 260.031,Z 455.296,A -85,B 0,C 180,E1 -18776.914,E2 -18776.914} C_VEL
LIN {X 0,Y 262.494,Z 468,A -85,B 0,C 180,E1 -18778.585,E2 -18778.585} C_VEL
LIN {X 0,Y 263.913,Z 479.578,A -85,B 0,C 180,E1 -18780.265,E2 -18780.265} C_VEL
LIN {X 0,Y 264.322,Z 485.468,A -85,B 0,C 180,E1 -18781.189,E2 -18781.189} C_VEL
LIN {X 0,Y 261.907,Z 496.843,A -85,B 0,C 180,E1 -18782.859,E2 -18782.859} C_VEL
LIN {X 0,Y 259.122,Z 507.294,A -85,B 0,C 180,E1 -18784.711,E2 -18784.711} C_VEL
LIN {X 0,Y 256.315,Z 517.693,A -85,B 0,C 180,E1 -18787,E2 -18787} C_VEL
LIN {X 0,Y 253.816,Z 526.273,A -85,B 0,C 180,E1 -18789.326,E2 -18789.326} C_VEL
LIN {X 0,Y 251.511,Z 534.486,A -85,B 0,C 180,E1 -18792.099,E2 -18792.099} C_VEL
LIN {X 0,Y 249.998,Z 540.241,A -85,B 0,C 180,E1 -18794.51,E2 -18794.51} C_VEL
LIN {X 0,Y 248.648,Z 544.952,A -85,B 0,C 180,E1 -18796.931,E2 -18796.931} C_VEL
LIN {X 0,Y 247.607,Z 549.836,A -85,B 0,C 180,E1 -18800.194,E2 -18800.194} C_VEL
LIN {X 0,Y 247.007,Z 553.231,A -85,B 0,C 180,E1 -18803.465,E2 -18803.465} C_VEL
LIN {X 0,Y 246.819,Z 555.238,A -85,B 0,C 180,E1 -18806.735,E2 -18806.735} C_VEL
LIN {X 0,Y 246.89,Z 555.9,A -85,B 0,C 180,E1 -18810,E2 -18810} C_VEL
LIN {X 0,Y 246.819,Z 555.224,A -85,B 0,C 180,E1 -18813.265,E2 -18813.265} C_VEL
LIN {X 0,Y 247.015,Z 553.206,A -85,B 0,C 180,E1 -18816.535,E2 -18816.535} C_VEL
LIN {X 0,Y 247.603,Z 549.797,A -85,B 0,C 180,E1 -18819.805,E2 -18819.805} C_VEL
LIN {X 0,Y 248.645,Z 544.893,A -85,B 0,C 180,E1 -18823.069,E2 -18823.069} C_VEL
LIN {X 0,Y 249.994,Z 540.166,A -85,B 0,C 180,E1 -18825.49,E2 -18825.49} C_VEL
LIN {X 0,Y 251.903,Z 532.888,A -85,B 0,C 180,E1 -18828.452,E2 -18828.452} C_VEL
LIN {X 0,Y 254.18,Z 524.804,A -85,B 0,C 180,E1 -18831.066,E2 -18831.066} C_VEL
LIN {X 0,Y 256.756,Z 515.928,A -85,B 0,C 180,E1 -18833.384,E2 -18833.384} C_VEL
LIN {X 0,Y 259.68,Z 505.176,A -85,B 0,C 180,E1 -18835.66,E2 -18835.66} C_VEL
LIN {X 0,Y 262.298,Z 494.851,A -85,B 0,C 180,E1 -18837.426,E2 -18837.426} C_VEL
LIN {X 0,Y 264.262,Z 485.227,A -85,B 0,C 180,E1 -18838.818,E2 -18838.818} C_VEL
LIN {X 0,Y 263.361,Z 474.454,A -85,B 0,C 180,E1 -18840.466,E2 -18840.466} C_VEL
LIN {X 0,Y 261.453,Z 462.389,A -85,B 0,C 180,E1 -18842.143,E2 -18842.143} C_VEL
LIN {X 0,Y 258.566,Z 449.891,A -85,B 0,C 180,E1 -18843.733,E2 -18843.733} C_VEL
LIN {X 0,Y 254.21,Z 436.367,A -85,B 0,C 180,E1 -18845.358,E2 -18845.358} C_VEL
LIN {X 0,Y 250.912,Z 428.281,A -85,B 0,C 180,E1 -18846.308,E2 -18846.308} C_VEL
LIN {X 0,Y 249.907,Z 425.002,A -85,B 0,C 180,E1 -18846.634,E2 -18846.634} C_VEL
LIN {X 0,Y 250.217,Z 421.781,A -85,B 0,C 180,E1 -18850.242,E2 -18850.242} C_VEL
LIN {X 0,Y 250.124,Z 419.404,A -85,B 0,C 180,E1 -18853.068,E2 -18853.068} C_VEL
LIN {X 0,Y 249.751,Z 416.329,A -85,B 0,C 180,E1 -18857.024,E2 -18857.024} C_VEL
LIN {X 0,Y 249.216,Z 413.025,A -85,B 0,C 180,E1 -18861.654,E2 -18861.654} C_VEL
LIN {X 0,Y 249.076,Z 412.086,A -85,B 0,C 180,E1 -18863.662,E2 -18863.662} C_VEL
LIN {X 0,Y 249.04,Z 412.091,A -85,B 0,C 180,E1 -18867.845,E2 -18867.845} C_VEL
LIN {X 0,Y 249.086,Z 412.084,A -85,B 0,C 180,E1 -18871.337,E2 -18871.337} C_VEL
LIN {X 0,Y 249.135,Z 412.078,A -85,B 0,C 180,E1 -18874.967,E2 -18874.967} C_VEL
LIN {X 0,Y 249.11,Z 412.08,A -85,B 0,C 180,E1 -18880.212,E2 -18880.212} C_VEL
LIN {X 0,Y 249.243,Z 412.064,A -85,B 0,C 180,E1 -18883.622,E2 -18883.622} C_VEL
LIN {X 0,Y 249.254,Z 412.058,A -85,B 0,C 180,E1 -18888.617,E2 -18888.617} C_VEL
LIN {X 0,Y 249.486,Z 412.03,A -85,B 0,C 180,E1 -18891.903,E2 -18891.903} C_VEL
LIN {X 0,Y 249.439,Z 412.041,A -85,B 0,C 180,E1 -18896.77,E2 -18896.77} C_VEL
LIN {X 0,Y 249.737,Z 412.002,A -85,B 0,C 180,E1 -18900,E2 -18900} C_VEL
LIN {X 0,Y 249.438,Z 412.041,A -85,B 0,C 180,E1 -18903.231,E2 -18903.231} C_VEL
LIN {X 0,Y 249.486,Z 412.034,A -85,B 0,C 180,E1 -18908.097,E2 -18908.097} C_VEL
LIN {X 0,Y 249.254,Z 412.063,A -85,B 0,C 180,E1 -18911.384,E2 -18911.384} C_VEL
LIN {X 0,Y 249.243,Z 412.06,A -85,B 0,C 180,E1 -18916.378,E2 -18916.378} C_VEL
LIN {X 0,Y 249.088,Z 412.083,A -85,B 0,C 180,E1 -18921.518,E2 -18921.518} C_VEL
LIN {X 0,Y 249.132,Z 412.078,A -85,B 0,C 180,E1 -18925.482,E2 -18925.482} C_VEL
LIN {X 0,Y 249.074,Z 412.085,A -85,B 0,C 180,E1 -18928.989,E2 -18928.989} C_VEL
LIN {X 0,Y 249.037,Z 412.09,A -85,B 0,C 180,E1 -18932.425,E2 -18932.425} C_VEL
LIN {X 0,Y 249.07,Z 412.086,A -85,B 0,C 180,E1 -18936.339,E2 -18936.339} C_VEL
LIN {X 0,Y 249.029,Z 412.092,A -85,B 0,C 180,E1 -18940.474,E2 -18940.474} C_VEL
LIN {X 0,Y 249.422,Z 414.896,A -85,B 0,C 180,E1 -18944.784,E2 -18944.784} C_VEL
LIN {X 0,Y 249.666,Z 416.822,A -85,B 0,C 180,E1 -18947.5,E2 -18947.5} C_VEL
LIN {X 0,Y 249.747,Z 418.431,A -85,B 0,C 180,E1 -18949.667,E2 -18949.667} C_VEL
LIN {X 0,Y 249.573,Z 421.543,A -85,B 0,C 180,E1 -18953.393,E2 -18953.393} C_VEL
LIN {X 0,Y 250.591,Z 424.571,A -85,B 0,C 180,E1 -18953.692,E2 -18953.692} C_VEL
LIN {X 0,Y 253.077,Z 430.03,A -85,B 0,C 180,E1 -18954.38,E2 -18954.38} C_VEL
LIN {X 0,Y 257.593,Z 442.231,A -85,B 0,C 180,E1 -18955.895,E2 -18955.895} C_VEL
LIN {X 0,Y 261.2,Z 454.955,A -85,B 0,C 180,E1 -18957.549,E2 -18957.549} C_VEL
LIN {X 0,Y 263.561,Z 467.204,A -85,B 0,C 180,E1 -18959.246,E2 -18959.246} C_VEL
LIN {X 0,Y 265.003,Z 479.095,A -85,B 0,C 180,E1 -18961.066,E2 -18961.066} C_VEL
LIN {X 0,Y 262.914,Z 489.528,A -85,B 0,C 180,E1 -18962.541,E2 -18962.541} C_VEL
LIN {X 0,Y 260.084,Z 500.427,A -85,B 0,C 180,E1 -18964.383,E2 -18964.383} C_VEL
LIN {X 0,Y 257.65,Z 509.556,A -85,B 0,C 180,E1 -18966.276,E2 -18966.276} C_VEL
LIN {X 0,Y 255.022,Z 518.703,A -85,B 0,C 180,E1 -18968.583,E2 -18968.583} C_VEL
LIN {X 0,Y 252.515,Z 527.45,A -85,B 0,C 180,E1 -18971.338,E2 -18971.338} C_VEL
LIN {X 0,Y 250.92,Z 533.587,A -85,B 0,C 180,E1 -18973.735,E2 -18973.735} C_VEL
LIN {X 0,Y 249.36,Z 538.674,A -85,B 0,C 180,E1 -18976.139,E2 -18976.139} C_VEL
LIN {X 0,Y 248.067,Z 543.942,A -85,B 0,C 180,E1 -18979.388,E2 -18979.388} C_VEL
LIN {X 0,Y 247.44,Z 546.882,A -85,B 0,C 180,E1 -18981.836,E2 -18981.836} C_VEL
LIN {X 0,Y 246.991,Z 549.581,A -85,B 0,C 180,E1 -18985.103,E2 -18985.103} C_VEL
LIN {X 0,Y 246.877,Z 550.93,A -85,B 0,C 180,E1 -18988.369,E2 -18988.369} C_VEL
LIN {X 0,Y 246.893,Z 551.108,A -85,B 0,C 180,E1 -18990,E2 -18990} C_VEL
LIN {X 0,Y 246.889,Z 550.476,A -85,B 0,C 180,E1 -18993.264,E2 -18993.264} C_VEL
LIN {X 0,Y 247.181,Z 548.508,A -85,B 0,C 180,E1 -18996.531,E2 -18996.531} C_VEL
LIN {X 0,Y 247.812,Z 545.158,A -85,B 0,C 180,E1 -18999.797,E2 -18999.797} C_VEL
LIN {X 0,Y 248.946,Z 540.327,A -85,B 0,C 180,E1 -19003.053,E2 -19003.053} C_VEL
LIN {X 0,Y 250.881,Z 533.856,A -85,B 0,C 180,E1 -19006.268,E2 -19006.268} C_VEL
LIN {X 0,Y 252.751,Z 526.788,A -85,B 0,C 180,E1 -19009.019,E2 -19009.019} C_VEL
LIN {X 0,Y 254.987,Z 519.103,A -85,B 0,C 180,E1 -19011.42,E2 -19011.42} C_VEL
LIN {X 0,Y 257.562,Z 510.035,A -85,B 0,C 180,E1 -19013.733,E2 -19013.733} C_VEL
LIN {X 0,Y 260.634,Z 499.048,A -85,B 0,C 180,E1 -19015.988,E2 -19015.988} C_VEL
LIN {X 0,Y 263.349,Z 487.839,A -85,B 0,C 180,E1 -19017.841,E2 -19017.841} C_VEL
LIN {X 0,Y 265.004,Z 479.926,A -85,B 0,C 180,E1 -19018.934,E2 -19018.934} C_VEL
LIN {X 0,Y 263.878,Z 469.141,A -85,B 0,C 180,E1 -19020.598,E2 -19020.598} C_VEL
LIN {X 0,Y 261.557,Z 456.323,A -85,B 0,C 180,E1 -19022.395,E2 -19022.395} C_VEL
LIN {X 0,Y 258.03,Z 443.769,A -85,B 0,C 180,E1 -19024.055,E2 -19024.055} C_VEL
LIN {X 0,Y 254.165,Z 432.648,A -85,B 0,C 180,E1 -19025.441,E2 -19025.441} C_VEL
LIN {X 0,Y 250.597,Z 424.481,A -85,B 0,C 180,E1 -19026.451,E2 -19026.451} C_VEL
LIN {X 0,Y 249.576,Z 421.356,A -85,B 0,C 180,E1 -19026.789,E2 -19026.789} C_VEL
LIN {X 0,Y 249.757,Z 418.369,A -85,B 0,C 180,E1 -19030.556,E2 -19030.556} C_VEL
LIN {X 0,Y 249.641,Z 416.606,A -85,B 0,C 180,E1 -19032.948,E2 -19032.948} C_VEL
LIN {X 0,Y 249.471,Z 414.993,A -85,B 0,C 180,E1 -19035.227,E2 -19035.227} C_VEL
LIN {X 0,Y 249.031,Z 412.093,A -85,B 0,C 180,E1 -19039.639,E2 -19039.639} C_VEL
LIN {X 0,Y 249.032,Z 412.089,A -85,B 0,C 180,E1 -19043.655,E2 -19043.655} C_VEL
LIN {X 0,Y 249.04,Z 412.087,A -85,B 0,C 180,E1 -19047.846,E2 -19047.846} C_VEL
LIN {X 0,Y 249.099,Z 412.082,A -85,B 0,C 180,E1 -19051.338,E2 -19051.338} C_VEL
LIN {X 0,Y 249.154,Z 412.075,A -85,B 0,C 180,E1 -19054.969,E2 -19054.969} C_VEL
LIN {X 0,Y 249.114,Z 412.074,A -85,B 0,C 180,E1 -19060.212,E2 -19060.212} C_VEL
LIN {X 0,Y 249.244,Z 412.065,A -85,B 0,C 180,E1 -19063.622,E2 -19063.622} C_VEL
LIN {X 0,Y 249.256,Z 412.061,A -85,B 0,C 180,E1 -19068.617,E2 -19068.617} C_VEL
LIN {X 0,Y 249.487,Z 412.033,A -85,B 0,C 180,E1 -19071.903,E2 -19071.903} C_VEL
LIN {X 0,Y 249.438,Z 412.039,A -85,B 0,C 180,E1 -19076.77,E2 -19076.77} C_VEL
LIN {X 0,Y 249.731,Z 412.004,A -85,B 0,C 180,E1 -19080,E2 -19080} C_VEL
LIN {X 0,Y 249.44,Z 412.038,A -85,B 0,C 180,E1 -19083.23,E2 -19083.23} C_VEL
LIN {X 0,Y 249.487,Z 412.032,A -85,B 0,C 180,E1 -19088.097,E2 -19088.097} C_VEL
LIN {X 0,Y 249.256,Z 412.064,A -85,B 0,C 180,E1 -19091.383,E2 -19091.383} C_VEL
LIN {X 0,Y 249.244,Z 412.063,A -85,B 0,C 180,E1 -19096.378,E2 -19096.378} C_VEL
LIN {X 0,Y 249.089,Z 412.083,A -85,B 0,C 180,E1 -19101.518,E2 -19101.518} C_VEL
LIN {X 0,Y 249.132,Z 412.077,A -85,B 0,C 180,E1 -19105.482,E2 -19105.482} C_VEL
LIN {X 0,Y 249.085,Z 412.084,A -85,B 0,C 180,E1 -19108.993,E2 -19108.993} C_VEL
LIN {X 0,Y 249.038,Z 412.091,A -85,B 0,C 180,E1 -19112.425,E2 -19112.425} C_VEL
LIN {X 0,Y 249.063,Z 412.088,A -85,B 0,C 180,E1 -19115.514,E2 -19115.514} C_VEL
LIN {X 0,Y 248.76,Z 412.273,A -85,B 0,C 180,E1 -19116.416,E2 -19116.416} C_VEL
LIN {X 0,Y 247.502,Z 413.076,A -85,B 0,C 180,E1 -19117.74,E2 -19117.74} C_VEL
LIN {X 0,Y 243.571,Z 415.879,A -85,B 0,C 180,E1 -19120.806,E2 -19120.806} C_VEL
LIN {X 0,Y 242.711,Z 417.027,A -85,B 0,C 180,E1 -19122.173,E2 -19122.173} C_VEL
LIN {X 0,Y 242.684,Z 417.374,A -85,B 0,C 180,E1 -19122.636,E2 -19122.636} C_VEL
LIN {X 0,Y 243.099,Z 420.102,A -85,B 0,C 180,E1 -19126.282,E2 -19126.282} C_VEL
LIN {X 0,Y 243.206,Z 422.032,A -85,B 0,C 180,E1 -19128.706,E2 -19128.706} C_VEL
LIN {X 0,Y 243.028,Z 424.978,A -85,B 0,C 180,E1 -19132.121,E2 -19132.121} C_VEL
LIN {X 0,Y 244.112,Z 428.205,A -85,B 0,C 180,E1 -19132.458,E2 -19132.458} C_VEL
LIN {X 0,Y 246.711,Z 434.45,A -85,B 0,C 180,E1 -19133.244,E2 -19133.244} C_VEL
LIN {X 0,Y 251.002,Z 446.725,A -85,B 0,C 180,E1 -19134.81,E2 -19134.81} C_VEL
LIN {X 0,Y 254.275,Z 458.974,A -85,B 0,C 180,E1 -19136.441,E2 -19136.441} C_VEL
LIN {X 0,Y 256.592,Z 472.379,A -85,B 0,C 180,E1 -19138.34,E2 -19138.34} C_VEL
LIN {X 0,Y 257.687,Z 484.103,A -85,B 0,C 180,E1 -19140.17,E2 -19140.17} C_VEL
LIN {X 0,Y 257.839,Z 486.826,A -85,B 0,C 180,E1 -19140.618,E2 -19140.618} C_VEL
LIN {X 0,Y 255.006,Z 499.037,A -85,B 0,C 180,E1 -19142.507,E2 -19142.507} C_VEL
LIN {X 0,Y 252.189,Z 509.118,A -85,B 0,C 180,E1 -19144.408,E2 -19144.408} C_VEL
LIN {X 0,Y 249.292,Z 519.142,A -85,B 0,C 180,E1 -19146.753,E2 -19146.753} C_VEL
LIN {X 0,Y 246.776,Z 527.467,A -85,B 0,C 180,E1 -19149.146,E2 -19149.146} C_VEL
LIN {X 0,Y 244.451,Z 535.428,A -85,B 0,C 180,E1 -19151.997,E2 -19151.997} C_VEL
LIN {X 0,Y 242.615,Z 541.838,A -85,B 0,C 180,E1 -19154.888,E2 -19154.888} C_VEL
LIN {X 0,Y 241.373,Z 546.276,A -85,B 0,C 180,E1 -19157.386,E2 -19157.386} C_VEL
LIN {X 0,Y 240.591,Z 549.768,A -85,B 0,C 180,E1 -19159.906,E2 -19159.906} C_VEL
LIN {X 0,Y 239.925,Z 553.162,A -85,B 0,C 180,E1 -19163.271,E2 -19163.271} C_VEL
LIN {X 0,Y 239.729,Z 555.169,A -85,B 0,C 180,E1 -19166.638,E2 -19166.638} C_VEL
LIN {X 0,Y 239.802,Z 555.831,A -85,B 0,C 180,E1 -19170,E2 -19170} C_VEL
LIN {X 0,Y 239.729,Z 555.155,A -85,B 0,C 180,E1 -19173.361,E2 -19173.361} C_VEL
LIN {X 0,Y 239.955,Z 553.137,A -85,B 0,C 180,E1 -19176.728,E2 -19176.728} C_VEL
LIN {X 0,Y 240.587,Z 549.727,A -85,B 0,C 180,E1 -19180.094,E2 -19180.094} C_VEL
LIN {X 0,Y 241.693,Z 544.822,A -85,B 0,C 180,E1 -19183.452,E2 -19183.452} C_VEL
LIN {X 0,Y 243.118,Z 540.096,A -85,B 0,C 180,E1 -19185.939,E2 -19185.939} C_VEL
LIN {X 0,Y 245.009,Z 533.283,A -85,B 0,C 180,E1 -19188.81,E2 -19188.81} C_VEL
LIN {X 0,Y 247.537,Z 524.733,A -85,B 0,C 180,E1 -19191.659,E2 -19191.659} C_VEL
LIN {X 0,Y 250.236,Z 515.857,A -85,B 0,C 180,E1 -19194.031,E2 -19194.031} C_VEL
LIN {X 0,Y 253.279,Z 505.104,A -85,B 0,C 180,E1 -19196.357,E2 -19196.357} C_VEL
LIN {X 0,Y 256.4,Z 493.384,A -85,B 0,C 180,E1 -19198.377,E2 -19198.377} C_VEL
LIN {X 0,Y 257.758,Z 486.58,A -85,B 0,C 180,E1 -19199.392,E2 -19199.392} C_VEL
LIN {X 0,Y 256.932,Z 475.227,A -85,B 0,C 180,E1 -19201.201,E2 -19201.201} C_VEL
LIN {X 0,Y 254.801,Z 461.926,A -85,B 0,C 180,E1 -19203.127,E2 -19203.127} C_VEL
LIN {X 0,Y 251.506,Z 448.484,A -85,B 0,C 180,E1 -19204.92,E2 -19204.92} C_VEL
LIN {X 0,Y 247.306,Z 435.999,A -85,B 0,C 180,E1 -19206.516,E2 -19206.516} C_VEL
LIN {X 0,Y 244.189,Z 428.395,A -85,B 0,C 180,E1 -19207.467,E2 -19207.467} C_VEL
LIN {X 0,Y 243.16,Z 425.719,A -85,B 0,C 180,E1 -19207.768,E2 -19207.768} C_VEL
LIN {X 0,Y 243.03,Z 424.89,A -85,B 0,C 180,E1 -19207.896,E2 -19207.896} C_VEL
LIN {X 0,Y 243.152,Z 421.69,A -85,B 0,C 180,E1 -19211.666,E2 -19211.666} C_VEL
LIN {X 0,Y 243.033,Z 419.882,A -85,B 0,C 180,E1 -19213.95,E2 -19213.95} C_VEL
LIN {X 0,Y 242.831,Z 418.061,A -85,B 0,C 180,E1 -19216.348,E2 -19216.348} C_VEL
LIN {X 0,Y 242.34,Z 415.234,A -85,B 0,C 180,E1 -19220.356,E2 -19220.356} C_VEL
LIN {X 0,Y 242.15,Z 413.839,A -85,B 0,C 180,E1 -19222.447,E2 -19222.447} C_VEL
LIN {X 0,Y 242.037,Z 412.964,A -85,B 0,C 180,E1 -19224.498,E2 -19224.498} C_VEL
LIN {X 0,Y 241.975,Z 412.971,A -85,B 0,C 180,E1 -19228.48,E2 -19228.48} C_VEL
LIN {X 0,Y 242.002,Z 412.968,A -85,B 0,C 180,E1 -19232.312,E2 -19232.312} C_VEL
LIN {X 0,Y 242.042,Z 412.962,A -85,B 0,C 180,E1 -19236.014,E2 -19236.014} C_VEL
LIN {X 0,Y 242.037,Z 412.961,A -85,B 0,C 180,E1 -19239.608,E2 -19239.608} C_VEL
LIN {X 0,Y 242.164,Z 412.945,A -85,B 0,C 180,E1 -19243.278,E2 -19243.278} C_VEL
LIN {X 0,Y 242.188,Z 412.939,A -85,B 0,C 180,E1 -19248.28,E2 -19248.28} C_VEL
LIN {X 0,Y 242.436,Z 412.91,A -85,B 0,C 180,E1 -19251.666,E2 -19251.666} C_VEL
LIN {X 0,Y 242.263,Z 412.935,A -85,B 0,C 180,E1 -19255.007,E2 -19255.007} C_VEL
LIN {X 0,Y 242.638,Z 412.886,A -85,B 0,C 180,E1 -19258.34,E2 -19258.34} C_VEL
LIN {X 0,Y 242.638,Z 412.886,A -85,B 0,C 180,E1 -19261.66,E2 -19261.66} C_VEL
LIN {X 0,Y 242.43,Z 412.911,A -85,B 0,C 180,E1 -19266.75,E2 -19266.75} C_VEL
LIN {X 0,Y 242.347,Z 412.922,A -85,B 0,C 180,E1 -19270.021,E2 -19270.021} C_VEL
LIN {X 0,Y 242.168,Z 412.945,A -85,B 0,C 180,E1 -19275.141,E2 -19275.141} C_VEL
LIN {X 0,Y 242.075,Z 412.957,A -85,B 0,C 180,E1 -19278.624,E2 -19278.624} C_VEL
LIN {X 0,Y 242.014,Z 412.964,A -85,B 0,C 180,E1 -19282.18,E2 -19282.18} C_VEL
LIN {X 0,Y 242.068,Z 412.957,A -85,B 0,C 180,E1 -19285.838,E2 -19285.838} C_VEL
LIN {X 0,Y 242.008,Z 412.965,A -85,B 0,C 180,E1 -19289.583,E2 -19289.583} C_VEL
LIN {X 0,Y 241.992,Z 412.967,A -85,B 0,C 180,E1 -19293.491,E2 -19293.491} C_VEL
LIN {X 0,Y 242.004,Z 412.965,A -85,B 0,C 180,E1 -19297.58,E2 -19297.58} C_VEL
LIN {X 0,Y 241.974,Z 412.969,A -85,B 0,C 180,E1 -19299.716,E2 -19299.716} C_VEL
LIN {X 0,Y 242.348,Z 415.678,A -85,B 0,C 180,E1 -19304.106,E2 -19304.106} C_VEL
LIN {X 0,Y 242.673,Z 418.52,A -85,B 0,C 180,E1 -19308.234,E2 -19308.234} C_VEL
LIN {X 0,Y 242.646,Z 421.649,A -85,B 0,C 180,E1 -19312.168,E2 -19312.168} C_VEL
LIN {X 0,Y 243.694,Z 424.632,A -85,B 0,C 180,E1 -19312.489,E2 -19312.489} C_VEL
LIN {X 0,Y 244.783,Z 426.827,A -85,B 0,C 180,E1 -19312.788,E2 -19312.788} C_VEL
LIN {X 0,Y 249.298,Z 437.787,A -85,B 0,C 180,E1 -19314.245,E2 -19314.245} C_VEL
LIN {X 0,Y 253.372,Z 450.538,A -85,B 0,C 180,E1 -19315.963,E2 -19315.963} C_VEL
LIN {X 0,Y 256.037,Z 461.895,A -85,B 0,C 180,E1 -19317.571,E2 -19317.571} C_VEL
LIN {X 0,Y 257.801,Z 473.143,A -85,B 0,C 180,E1 -19319.275,E2 -19319.275} C_VEL
LIN {X 0,Y 258.525,Z 480.316,A -85,B 0,C 180,E1 -19320.45,E2 -19320.45} C_VEL
LIN {X 0,Y 256.596,Z 489.736,A -85,B 0,C 180,E1 -19321.831,E2 -19321.831} C_VEL
LIN {X 0,Y 253.702,Z 500.499,A -85,B 0,C 180,E1 -19323.69,E2 -19323.69} C_VEL
LIN {X 0,Y 251.133,Z 509.628,A -85,B 0,C 180,E1 -19325.62,E2 -19325.62} C_VEL
LIN {X 0,Y 248.398,Z 518.775,A -85,B 0,C 180,E1 -19327.983,E2 -19327.983} C_VEL
LIN {X 0,Y 245.901,Z 526.941,A -85,B 0,C 180,E1 -19330.59,E2 -19330.59} C_VEL
LIN {X 0,Y 244.095,Z 533.658,A -85,B 0,C 180,E1 -19333.267,E2 -19333.267} C_VEL
LIN {X 0,Y 242.016,Z 540.184,A -85,B 0,C 180,E1 -19336.567,E2 -19336.567} C_VEL
LIN {X 0,Y 240.792,Z 545.073,A -85,B 0,C 180,E1 -19339.914,E2 -19339.914} C_VEL
LIN {X 0,Y 240.103,Z 548.473,A -85,B 0,C 180,E1 -19343.276,E2 -19343.276} C_VEL
LIN {X 0,Y 239.799,Z 550.49,A -85,B 0,C 180,E1 -19346.64,E2 -19346.64} C_VEL
LIN {X 0,Y 239.806,Z 551.177,A -85,B 0,C 180,E1 -19350,E2 -19350} C_VEL
LIN {X 0,Y 239.799,Z 550.545,A -85,B 0,C 180,E1 -19353.361,E2 -19353.361} C_VEL
LIN {X 0,Y 240.101,Z 548.576,A -85,B 0,C 180,E1 -19356.724,E2 -19356.724} C_VEL
LIN {X 0,Y 240.778,Z 545.227,A -85,B 0,C 180,E1 -19360.087,E2 -19360.087} C_VEL
LIN {X 0,Y 241.993,Z 540.395,A -85,B 0,C 180,E1 -19363.435,E2 -19363.435} C_VEL
LIN {X 0,Y 244.053,Z 533.924,A -85,B 0,C 180,E1 -19366.737,E2 -19366.737} C_VEL
LIN {X 0,Y 245.874,Z 527.317,A -85,B 0,C 180,E1 -19369.393,E2 -19369.393} C_VEL
LIN {X 0,Y 248.354,Z 519.17,A -85,B 0,C 180,E1 -19372.022,E2 -19372.022} C_VEL
LIN {X 0,Y 251.063,Z 510.102,A -85,B 0,C 180,E1 -19374.387,E2 -19374.387} C_VEL
LIN {X 0,Y 254.249,Z 499.114,A -85,B 0,C 180,E1 -19376.692,E2 -19376.692} C_VEL
LIN {X 0,Y 257.042,Z 488.087,A -85,B 0,C 180,E1 -19378.554,E2 -19378.554} C_VEL
LIN {X 0,Y 258.553,Z 481.047,A -85,B 0,C 180,E1 -19379.561,E2 -19379.561} C_VEL
LIN {X 0,Y 257.342,Z 469.58,A -85,B 0,C 180,E1 -19381.414,E2 -19381.414} C_VEL
LIN {X 0,Y 255.12,Z 457.072,A -85,B 0,C 180,E1 -19383.245,E2 -19383.245} C_VEL
LIN {X 0,Y 251.3,Z 443.499,A -85,B 0,C 180,E1 -19385.126,E2 -19385.126} C_VEL
LIN {X 0,Y 247.029,Z 432,A -85,B 0,C 180,E1 -19386.668,E2 -19386.668} C_VEL
LIN {X 0,Y 244.051,Z 425.223,A -85,B 0,C 180,E1 -19387.565,E2 -19387.565} C_VEL
LIN {X 0,Y 242.712,Z 422.071,A -85,B 0,C 180,E1 -19387.946,E2 -19387.946} C_VEL
LIN {X 0,Y 242.611,Z 421.385,A -85,B 0,C 180,E1 -19388.088,E2 -19388.088} C_VEL
LIN {X 0,Y 242.678,Z 418.631,A -85,B 0,C 180,E1 -19391.766,E2 -19391.766} C_VEL
LIN {X 0,Y 242.376,Z 415.773,A -85,B 0,C 180,E1 -19395.9,E2 -19395.9} C_VEL
LIN {X 0,Y 241.972,Z 413,A -85,B 0,C 180,E1 -19400.284,E2 -19400.284} C_VEL
LIN {X 0,Y 241.984,Z 412.968,A -85,B 0,C 180,E1 -19404.488,E2 -19404.488} C_VEL
LIN {X 0,Y 241.977,Z 412.967,A -85,B 0,C 180,E1 -19408.48,E2 -19408.48} C_VEL
LIN {X 0,Y 242.012,Z 412.965,A -85,B 0,C 180,E1 -19412.313,E2 -19412.313} C_VEL
LIN {X 0,Y 242.06,Z 412.954,A -85,B 0,C 180,E1 -19416.016,E2 -19416.016} C_VEL
LIN {X 0,Y 242.04,Z 412.954,A -85,B 0,C 180,E1 -19419.608,E2 -19419.608} C_VEL
LIN {X 0,Y 242.166,Z 412.945,A -85,B 0,C 180,E1 -19423.278,E2 -19423.278} C_VEL
LIN {X 0,Y 242.189,Z 412.943,A -85,B 0,C 180,E1 -19428.28,E2 -19428.28} C_VEL
LIN {X 0,Y 242.438,Z 412.91,A -85,B 0,C 180,E1 -19431.666,E2 -19431.666} C_VEL
LIN {X 0,Y 242.263,Z 412.934,A -85,B 0,C 180,E1 -19435.007,E2 -19435.007} C_VEL
LIN {X 0,Y 242.639,Z 412.885,A -85,B 0,C 180,E1 -19438.34,E2 -19438.34} C_VEL
LIN {X 0,Y 242.64,Z 412.886,A -85,B 0,C 180,E1 -19441.66,E2 -19441.66} C_VEL
LIN {X 0,Y 242.437,Z 412.913,A -85,B 0,C 180,E1 -19446.659,E2 -19446.659} C_VEL
LIN {X 0,Y 242.348,Z 412.921,A -85,B 0,C 180,E1 -19450.02,E2 -19450.02} C_VEL
LIN {X 0,Y 242.169,Z 412.944,A -85,B 0,C 180,E1 -19455.141,E2 -19455.141} C_VEL
LIN {X 0,Y 242.076,Z 412.956,A -85,B 0,C 180,E1 -19458.624,E2 -19458.624} C_VEL
LIN {X 0,Y 242.015,Z 412.965,A -85,B 0,C 180,E1 -19462.18,E2 -19462.18} C_VEL
LIN {X 0,Y 242.068,Z 412.958,A -85,B 0,C 180,E1 -19465.838,E2 -19465.838} C_VEL
LIN {X 0,Y 242.032,Z 412.958,A -85,B 0,C 180,E1 -19469.58,E2 -19469.58} C_VEL
LIN {X 0,Y 241.993,Z 412.969,A -85,B 0,C 180,E1 -19473.491,E2 -19473.491} C_VEL
LIN {X 0,Y 242.03,Z 412.966,A -85,B 0,C 180,E1 -19475.604,E2 -19475.604} C_VEL
LIN {X 0,Y 242.248,Z 414.473,A -85,B 0,C 180,E1 -19478.435,E2 -19478.435} C_VEL
LIN {X 0,Y 242.684,Z 417.374,A -85,B 0,C 180,E1 -19482.636,E2 -19482.636} C_VEL
LIN {X 0,Y 242.18,Z 418.488,A -85,B 0,C 180,E1 -19484,E2 -19484} C_VEL
LIN {X 0,Y 239.553,Z 420.645,A -85,B 0,C 180,E1 -19486.215,E2 -19486.215} C_VEL
LIN {X 0,Y 236.436,Z 423.303,A -85,B 0,C 180,E1 -19488.941,E2 -19488.941} C_VEL
LIN {X 0,Y 236.105,Z 424.116,A -85,B 0,C 180,E1 -19489.887,E2 -19489.887} C_VEL
LIN {X 0,Y 236.117,Z 425.076,A -85,B 0,C 180,E1 -19490.812,E2 -19490.812} C_VEL
LIN {X 0,Y 237.208,Z 428.158,A -85,B 0,C 180,E1 -19491.166,E2 -19491.166} C_VEL
LIN {X 0,Y 238.299,Z 430.298,A -85,B 0,C 180,E1 -19491.478,E2 -19491.478} C_VEL
LIN {X 0,Y 242.961,Z 442.301,A -85,B 0,C 180,E1 -19493.109,E2 -19493.109} C_VEL
LIN {X 0,Y 246.449,Z 453.952,A -85,B 0,C 180,E1 -19494.716,E2 -19494.716} C_VEL
LIN {X 0,Y 248.984,Z 465.462,A -85,B 0,C 180,E1 -19496.374,E2 -19496.374} C_VEL
LIN {X 0,Y 250.657,Z 477.722,A -85,B 0,C 180,E1 -19498.264,E2 -19498.264} C_VEL
LIN {X 0,Y 251.358,Z 488.113,A -85,B 0,C 180,E1 -19500.021,E2 -19500.021} C_VEL
LIN {X 0,Y 248.415,Z 500.041,A -85,B 0,C 180,E1 -19501.943,E2 -19501.943} C_VEL
LIN {X 0,Y 245.246,Z 510.835,A -85,B 0,C 180,E1 -19504.086,E2 -19504.086} C_VEL
LIN {X 0,Y 242.286,Z 520.563,A -85,B 0,C 180,E1 -19506.494,E2 -19506.494} C_VEL
LIN {X 0,Y 239.725,Z 528.633,A -85,B 0,C 180,E1 -19508.953,E2 -19508.953} C_VEL
LIN {X 0,Y 237.692,Z 535.007,A -85,B 0,C 180,E1 -19511.311,E2 -19511.311} C_VEL
LIN {X 0,Y 235.737,Z 541.77,A -85,B 0,C 180,E1 -19514.436,E2 -19514.436} C_VEL
LIN {X 0,Y 234.102,Z 547.452,A -85,B 0,C 180,E1 -19517.869,E2 -19517.869} C_VEL
LIN {X 0,Y 233.17,Z 551.575,A -85,B 0,C 180,E1 -19521.332,E2 -19521.332} C_VEL
LIN {X 0,Y 232.729,Z 554.267,A -85,B 0,C 180,E1 -19524.802,E2 -19524.802} C_VEL
LIN {X 0,Y 232.665,Z 555.599,A -85,B 0,C 180,E1 -19528.269,E2 -19528.269} C_VEL
LIN {X 0,Y 232.717,Z 555.762,A -85,B 0,C 180,E1 -19530,E2 -19530} C_VEL
LIN {X 0,Y 232.641,Z 555.086,A -85,B 0,C 180,E1 -19533.464,E2 -19533.464} C_VEL
LIN {X 0,Y 232.891,Z 553.067,A -85,B 0,C 180,E1 -19536.933,E2 -19536.933} C_VEL
LIN {X 0,Y 233.556,Z 549.656,A -85,B 0,C 180,E1 -19540.402,E2 -19540.402} C_VEL
LIN {X 0,Y 234.76,Z 544.752,A -85,B 0,C 180,E1 -19543.857,E2 -19543.857} C_VEL
LIN {X 0,Y 236.261,Z 540.025,A -85,B 0,C 180,E1 -19546.415,E2 -19546.415} C_VEL
LIN {X 0,Y 238.129,Z 533.672,A -85,B 0,C 180,E1 -19549.191,E2 -19549.191} C_VEL
LIN {X 0,Y 240.504,Z 526.018,A -85,B 0,C 180,E1 -19551.875,E2 -19551.875} C_VEL
LIN {X 0,Y 243.233,Z 517.414,A -85,B 0,C 180,E1 -19554.314,E2 -19554.314} C_VEL
LIN {X 0,Y 246.343,Z 506.986,A -85,B 0,C 180,E1 -19556.701,E2 -19556.701} C_VEL
LIN {X 0,Y 249.304,Z 496.497,A -85,B 0,C 180,E1 -19558.635,E2 -19558.635} C_VEL
LIN {X 0,Y 251.286,Z 487.826,A -85,B 0,C 180,E1 -19559.998,E2 -19559.998} C_VEL
LIN {X 0,Y 250.498,Z 476.407,A -85,B 0,C 180,E1 -19561.911,E2 -19561.911} C_VEL
LIN {X 0,Y 248.567,Z 463.313,A -85,B 0,C 180,E1 -19563.904,E2 -19563.904} C_VEL
LIN {X 0,Y 245.96,Z 452.267,A -85,B 0,C 180,E1 -19565.475,E2 -19565.475} C_VEL
LIN {X 0,Y 242.124,Z 440.009,A -85,B 0,C 180,E1 -19567.148,E2 -19567.148} C_VEL
LIN {X 0,Y 237.733,Z 429.01,A -85,B 0,C 180,E1 -19568.637,E2 -19568.637} C_VEL
LIN {X 0,Y 236.254,Z 425.837,A -85,B 0,C 180,E1 -19569.067,E2 -19569.067} C_VEL
LIN {X 0,Y 236.071,Z 424.843,A -85,B 0,C 180,E1 -19569.175,E2 -19569.175} C_VEL
LIN {X 0,Y 236.124,Z 422.624,A -85,B 0,C 180,E1 -19571.918,E2 -19571.918} C_VEL
LIN {X 0,Y 235.878,Z 419.791,A -85,B 0,C 180,E1 -19575.65,E2 -19575.65} C_VEL
LIN {X 0,Y 235.525,Z 417.467,A -85,B 0,C 180,E1 -19578.969,E2 -19578.969} C_VEL
LIN {X 0,Y 235.092,Z 414.669,A -85,B 0,C 180,E1 -19583.281,E2 -19583.281} C_VEL
LIN {X 0,Y 234.961,Z 413.845,A -85,B 0,C 180,E1 -19585.367,E2 -19585.367} C_VEL
LIN {X 0,Y 234.923,Z 413.85,A -85,B 0,C 180,E1 -19589.431,E2 -19589.431} C_VEL
LIN {X 0,Y 234.994,Z 413.84,A -85,B 0,C 180,E1 -19593.794,E2 -19593.794} C_VEL
LIN {X 0,Y 234.999,Z 413.839,A -85,B 0,C 180,E1 -19598.969,E2 -19598.969} C_VEL
LIN {X 0,Y 235.097,Z 413.824,A -85,B 0,C 180,E1 -19603.059,E2 -19603.059} C_VEL
LIN {X 0,Y 235.148,Z 413.819,A -85,B 0,C 180,E1 -19607.924,E2 -19607.924} C_VEL
LIN {X 0,Y 235.392,Z 413.789,A -85,B 0,C 180,E1 -19611.415,E2 -19611.415} C_VEL
LIN {X 0,Y 235.407,Z 413.78,A -85,B 0,C 180,E1 -19613.142,E2 -19613.142} C_VEL
LIN {X 0,Y 235.598,Z 413.763,A -85,B 0,C 180,E1 -19618.291,E2 -19618.291} C_VEL
LIN {X 0,Y 235.597,Z 413.763,A -85,B 0,C 180,E1 -19621.71,E2 -19621.71} C_VEL
LIN {X 0,Y 235.407,Z 413.787,A -85,B 0,C 180,E1 -19626.859,E2 -19626.859} C_VEL
LIN {X 0,Y 235.255,Z 413.805,A -85,B 0,C 180,E1 -19630.326,E2 -19630.326} C_VEL
LIN {X 0,Y 235.115,Z 413.824,A -85,B 0,C 180,E1 -19635.606,E2 -19635.606} C_VEL
LIN {X 0,Y 235.011,Z 413.838,A -85,B 0,C 180,E1 -19639.206,E2 -19639.206} C_VEL
LIN {X 0,Y 234.962,Z 413.842,A -85,B 0,C 180,E1 -19642.883,E2 -19642.883} C_VEL
LIN {X 0,Y 234.969,Z 413.842,A -85,B 0,C 180,E1 -19646.658,E2 -19646.658} C_VEL
LIN {X 0,Y 234.924,Z 413.848,A -85,B 0,C 180,E1 -19650.569,E2 -19650.569} C_VEL
LIN {X 0,Y 234.962,Z 413.843,A -85,B 0,C 180,E1 -19654.633,E2 -19654.633} C_VEL
LIN {X 0,Y 234.943,Z 413.846,A -85,B 0,C 180,E1 -19658.945,E2 -19658.945} C_VEL
LIN {X 0,Y 235.3,Z 416.454,A -85,B 0,C 180,E1 -19663.391,E2 -19663.391} C_VEL
LIN {X 0,Y 235.572,Z 418.6,A -85,B 0,C 180,E1 -19666.672,E2 -19666.672} C_VEL
LIN {X 0,Y 235.646,Z 420.952,A -85,B 0,C 180,E1 -19670.012,E2 -19670.012} C_VEL
LIN {X 0,Y 235.671,Z 421.731,A -85,B 0,C 180,E1 -19670.837,E2 -19670.837} C_VEL
LIN {X 0,Y 236.733,Z 424.714,A -85,B 0,C 180,E1 -19671.183,E2 -19671.183} C_VEL
LIN {X 0,Y 237.937,Z 426.918,A -85,B 0,C 180,E1 -19671.525,E2 -19671.525} C_VEL
LIN {X 0,Y 242.533,Z 437.736,A -85,B 0,C 180,E1 -19673.075,E2 -19673.075} C_VEL
LIN {X 0,Y 245.958,Z 447.912,A -85,B 0,C 180,E1 -19674.524,E2 -19674.524} C_VEL
LIN {X 0,Y 249.134,Z 460.07,A -85,B 0,C 180,E1 -19676.323,E2 -19676.323} C_VEL
LIN {X 0,Y 251.164,Z 472.404,A -85,B 0,C 180,E1 -19678.248,E2 -19678.248} C_VEL
LIN {X 0,Y 252.086,Z 482.005,A -85,B 0,C 180,E1 -19679.879,E2 -19679.879} C_VEL
LIN {X 0,Y 249.485,Z 493.189,A -85,B 0,C 180,E1 -19681.617,E2 -19681.617} C_VEL
LIN {X 0,Y 246.213,Z 504.436,A -85,B 0,C 180,E1 -19683.741,E2 -19683.741} C_VEL
LIN {X 0,Y 243.258,Z 514.484,A -85,B 0,C 180,E1 -19686.142,E2 -19686.142} C_VEL
LIN {X 0,Y 240.534,Z 522.828,A -85,B 0,C 180,E1 -19688.578,E2 -19688.578} C_VEL
LIN {X 0,Y 238.062,Z 530.795,A -85,B 0,C 180,E1 -19691.497,E2 -19691.497} C_VEL
LIN {X 0,Y 236.654,Z 535.532,A -85,B 0,C 180,E1 -19693.613,E2 -19693.613} C_VEL
LIN {X 0,Y 235.08,Z 540.254,A -85,B 0,C 180,E1 -19696.163,E2 -19696.163} C_VEL
LIN {X 0,Y 233.78,Z 545.143,A -85,B 0,C 180,E1 -19699.609,E2 -19699.609} C_VEL
LIN {X 0,Y 233.052,Z 548.543,A -85,B 0,C 180,E1 -19703.072,E2 -19703.072} C_VEL
LIN {X 0,Y 232.712,Z 550.559,A -85,B 0,C 180,E1 -19706.537,E2 -19706.537} C_VEL
LIN {X 0,Y 232.721,Z 551.246,A -85,B 0,C 180,E1 -19710,E2 -19710} C_VEL
LIN {X 0,Y 232.712,Z 550.613,A -85,B 0,C 180,E1 -19713.463,E2 -19713.463} C_VEL
LIN {X 0,Y 233.05,Z 548.645,A -85,B 0,C 180,E1 -19716.928,E2 -19716.928} C_VEL
LIN {X 0,Y 233.762,Z 545.295,A -85,B 0,C 180,E1 -19720.393,E2 -19720.393} C_VEL
LIN {X 0,Y 235.057,Z 540.463,A -85,B 0,C 180,E1 -19723.839,E2 -19723.839} C_VEL
LIN {X 0,Y 237.218,Z 533.992,A -85,B 0,C 180,E1 -19727.234,E2 -19727.234} C_VEL
LIN {X 0,Y 239.202,Z 527.263,A -85,B 0,C 180,E1 -19730.005,E2 -19730.005} C_VEL
LIN {X 0,Y 241.775,Z 519.237,A -85,B 0,C 180,E1 -19732.654,E2 -19732.654} C_VEL
LIN {X 0,Y 244.607,Z 510.168,A -85,B 0,C 180,E1 -19735.075,E2 -19735.075} C_VEL
LIN {X 0,Y 247.91,Z 499.179,A -85,B 0,C 180,E1 -19737.431,E2 -19737.431} C_VEL
LIN {X 0,Y 250.695,Z 488.63,A -85,B 0,C 180,E1 -19739.257,E2 -19739.257} C_VEL
LIN {X 0,Y 252.114,Z 482.235,A -85,B 0,C 180,E1 -19740.212,E2 -19740.212} C_VEL
LIN {X 0,Y 250.978,Z 470.837,A -85,B 0,C 180,E1 -19742.144,E2 -19742.144} C_VEL
LIN {X 0,Y 248.915,Z 458.827,A -85,B 0,C 180,E1 -19744.001,E2 -19744.001} C_VEL
LIN {X 0,Y 245.567,Z 446.384,A -85,B 0,C 180,E1 -19745.832,E2 -19745.832} C_VEL
LIN {X 0,Y 241.481,Z 435.02,A -85,B 0,C 180,E1 -19747.454,E2 -19747.454} C_VEL
LIN {X 0,Y 237.271,Z 425.564,A -85,B 0,C 180,E1 -19748.822,E2 -19748.822} C_VEL
LIN {X 0,Y 235.88,Z 422.72,A -85,B 0,C 180,E1 -19749.225,E2 -19749.225} C_VEL
LIN {X 0,Y 235.636,Z 421.496,A -85,B 0,C 180,E1 -19749.395,E2 -19749.395} C_VEL
LIN {X 0,Y 235.679,Z 419.755,A -85,B 0,C 180,E1 -19751.797,E2 -19751.797} C_VEL
LIN {X 0,Y 235.408,Z 417.098,A -85,B 0,C 180,E1 -19755.767,E2 -19755.767} C_VEL
LIN {X 0,Y 235.107,Z 415.152,A -85,B 0,C 180,E1 -19758.879,E2 -19758.879} C_VEL
LIN {X 0,Y 234.925,Z 413.854,A -85,B 0,C 180,E1 -19761.08,E2 -19761.08} C_VEL
LIN {X 0,Y 234.929,Z 413.846,A -85,B 0,C 180,E1 -19765.362,E2 -19765.362} C_VEL
LIN {X 0,Y 234.934,Z 413.847,A -85,B 0,C 180,E1 -19769.432,E2 -19769.432} C_VEL
LIN {X 0,Y 234.997,Z 413.839,A -85,B 0,C 180,E1 -19773.794,E2 -19773.794} C_VEL
LIN {X 0,Y 235.014,Z 413.831,A -85,B 0,C 180,E1 -19778.97,E2 -19778.97} C_VEL
LIN {X 0,Y 235.099,Z 413.825,A -85,B 0,C 180,E1 -19783.059,E2 -19783.059} C_VEL
LIN {X 0,Y 235.15,Z 413.819,A -85,B 0,C 180,E1 -19787.924,E2 -19787.924} C_VEL
LIN {X 0,Y 235.393,Z 413.786,A -85,B 0,C 180,E1 -19791.415,E2 -19791.415} C_VEL
LIN {X 0,Y 235.409,Z 413.786,A -85,B 0,C 180,E1 -19793.141,E2 -19793.141} C_VEL
LIN {X 0,Y 235.598,Z 413.762,A -85,B 0,C 180,E1 -19798.29,E2 -19798.29} C_VEL
LIN {X 0,Y 235.599,Z 413.763,A -85,B 0,C 180,E1 -19801.709,E2 -19801.709} C_VEL
LIN {X 0,Y 235.409,Z 413.788,A -85,B 0,C 180,E1 -19806.858,E2 -19806.858} C_VEL
LIN {X 0,Y 235.256,Z 413.804,A -85,B 0,C 180,E1 -19810.326,E2 -19810.326} C_VEL
LIN {X 0,Y 235.116,Z 413.823,A -85,B 0,C 180,E1 -19815.606,E2 -19815.606} C_VEL
LIN {X 0,Y 235.011,Z 413.835,A -85,B 0,C 180,E1 -19819.205,E2 -19819.205} C_VEL
LIN {X 0,Y 234.963,Z 413.839,A -85,B 0,C 180,E1 -19822.882,E2 -19822.882} C_VEL
LIN {X 0,Y 234.972,Z 413.837,A -85,B 0,C 180,E1 -19826.657,E2 -19826.657} C_VEL
LIN {X 0,Y 234.934,Z 413.843,A -85,B 0,C 180,E1 -19830.567,E2 -19830.567} C_VEL
LIN {X 0,Y 234.962,Z 413.846,A -85,B 0,C 180,E1 -19834.633,E2 -19834.633} C_VEL
LIN {X 0,Y 235.1,Z 414.722,A -85,B 0,C 180,E1 -19836.718,E2 -19836.718} C_VEL
LIN {X 0,Y 235.649,Z 418.029,A -85,B 0,C 180,E1 -19841.789,E2 -19841.789} C_VEL
LIN {X 0,Y 236.008,Z 420.775,A -85,B 0,C 180,E1 -19845.617,E2 -19845.617} C_VEL
LIN {X 0,Y 236.16,Z 423.474,A -85,B 0,C 180,E1 -19849.102,E2 -19849.102} C_VEL
LIN {X 0,Y 236.105,Z 424.116,A -85,B 0,C 180,E1 -19849.887,E2 -19849.887} C_VEL
LIN {X 0,Y 236.369,Z 425.192,A -85,B 0,C 180,E1 -19850.49,E2 -19850.49} C_VEL
LIN {X 0,Y 237.248,Z 427.717,A -85,B 0,C 180,E1 -19851.113,E2 -19851.113} C_VEL
LIN {X 0,Y 238.595,Z 431.892,A -85,B 0,C 180,E1 -19851.628,E2 -19851.628} C_VEL
LIN {X 0,Y 239.302,Z 437.742,A -85,B 0,C 180,E1 -19852.098,E2 -19852.098} C_VEL
LIN {X 0,Y 238.974,Z 448.306,A -85,B 0,C 180,E1 -19852.888,E2 -19852.888} C_VEL
LIN {X 0,Y 239.443,Z 452.197,A -85,B 0,C 180,E1 -19853.352,E2 -19853.352} C_VEL
LIN {X 0,Y 242.32,Z 464.378,A -85,B 0,C 180,E1 -19855.192,E2 -19855.192} C_VEL
LIN {X 0,Y 244.075,Z 476.741,A -85,B 0,C 180,E1 -19857.162,E2 -19857.162} C_VEL
LIN {X 0,Y 244.856,Z 488.391,A -85,B 0,C 180,E1 -19859.203,E2 -19859.203} C_VEL
LIN {X 0,Y 244.087,Z 492.785,A -85,B 0,C 180,E1 -19859.914,E2 -19859.914} C_VEL
LIN {X 0,Y 241.231,Z 503.178,A -85,B 0,C 180,E1 -19861.743,E2 -19861.743} C_VEL
LIN {X 0,Y 238.268,Z 512.551,A -85,B 0,C 180,E1 -19863.74,E2 -19863.74} C_VEL
LIN {X 0,Y 235.285,Z 521.982,A -85,B 0,C 180,E1 -19866.218,E2 -19866.218} C_VEL
LIN {X 0,Y 232.269,Z 530.963,A -85,B 0,C 180,E1 -19869.174,E2 -19869.174} C_VEL
LIN {X 0,Y 230.523,Z 536.433,A -85,B 0,C 180,E1 -19871.389,E2 -19871.389} C_VEL
LIN {X 0,Y 228.877,Z 541.702,A -85,B 0,C 180,E1 -19873.957,E2 -19873.957} C_VEL
LIN {X 0,Y 227.105,Z 547.384,A -85,B 0,C 180,E1 -19877.489,E2 -19877.489} C_VEL
LIN {X 0,Y 226.125,Z 551.507,A -85,B 0,C 180,E1 -19881.06,E2 -19881.06} C_VEL
LIN {X 0,Y 225.645,Z 554.199,A -85,B 0,C 180,E1 -19884.638,E2 -19884.638} C_VEL
LIN {X 0,Y 225.565,Z 555.53,A -85,B 0,C 180,E1 -19888.214,E2 -19888.214} C_VEL
LIN {X 0,Y 225.633,Z 555.693,A -85,B 0,C 180,E1 -19890,E2 -19890} C_VEL
LIN {X 0,Y 225.541,Z 555.017,A -85,B 0,C 180,E1 -19893.573,E2 -19893.573} C_VEL
LIN {X 0,Y 225.822,Z 552.998,A -85,B 0,C 180,E1 -19897.151,E2 -19897.151} C_VEL
LIN {X 0,Y 226.545,Z 549.587,A -85,B 0,C 180,E1 -19900.727,E2 -19900.727} C_VEL
LIN {X 0,Y 227.846,Z 544.682,A -85,B 0,C 180,E1 -19904.286,E2 -19904.286} C_VEL
LIN {X 0,Y 229.41,Z 539.954,A -85,B 0,C 180,E1 -19906.92,E2 -19906.92} C_VEL
LIN {X 0,Y 231.516,Z 533.212,A -85,B 0,C 180,E1 -19909.922,E2 -19909.922} C_VEL
LIN {X 0,Y 233.882,Z 525.947,A -85,B 0,C 180,E1 -19912.527,E2 -19912.527} C_VEL
LIN {X 0,Y 236.768,Z 517.343,A -85,B 0,C 180,E1 -19915.023,E2 -19915.023} C_VEL
LIN {X 0,Y 239.41,Z 508.819,A -85,B 0,C 180,E1 -19917.066,E2 -19917.066} C_VEL
LIN {X 0,Y 242.775,Z 497.599,A -85,B 0,C 180,E1 -19919.242,E2 -19919.242} C_VEL
LIN {X 0,Y 244.722,Z 489.807,A -85,B 0,C 180,E1 -19920.509,E2 -19920.509} C_VEL
LIN {X 0,Y 244.456,Z 481.09,A -85,B 0,C 180,E1 -19922.063,E2 -19922.063} C_VEL
LIN {X 0,Y 242.889,Z 468.233,A -85,B 0,C 180,E1 -19924.179,E2 -19924.179} C_VEL
LIN {X 0,Y 240.295,Z 455.621,A -85,B 0,C 180,E1 -19926.102,E2 -19926.102} C_VEL
LIN {X 0,Y 236.494,Z 442.903,A -85,B 0,C 180,E1 -19927.969,E2 -19927.969} C_VEL
LIN {X 0,Y 232.745,Z 433.131,A -85,B 0,C 180,E1 -19929.381,E2 -19929.381} C_VEL
LIN {X 0,Y 230.679,Z 428.79,A -85,B 0,C 180,E1 -19930.056,E2 -19930.056} C_VEL
LIN {X 0,Y 229.252,Z 425.566,A -85,B 0,C 180,E1 -19930.51,E2 -19930.51} C_VEL
LIN {X 0,Y 229.095,Z 424.759,A -85,B 0,C 180,E1 -19930.621,E2 -19930.621} C_VEL
LIN {X 0,Y 229.081,Z 423.244,A -85,B 0,C 180,E1 -19932.583,E2 -19932.583} C_VEL
LIN {X 0,Y 228.907,Z 421.408,A -85,B 0,C 180,E1 -19935.077,E2 -19935.077} C_VEL
LIN {X 0,Y 228.698,Z 419.713,A -85,B 0,C 180,E1 -19937.521,E2 -19937.521} C_VEL
LIN {X 0,Y 228.22,Z 416.821,A -85,B 0,C 180,E1 -19941.983,E2 -19941.983} C_VEL
LIN {X 0,Y 228.028,Z 415.515,A -85,B 0,C 180,E1 -19944.155,E2 -19944.155} C_VEL
LIN {X 0,Y 227.891,Z 414.726,A -85,B 0,C 180,E1 -19946.373,E2 -19946.373} C_VEL
LIN {X 0,Y 227.905,Z 414.723,A -85,B 0,C 180,E1 -19950.436,E2 -19950.436} C_VEL
LIN {X 0,Y 227.925,Z 414.72,A -85,B 0,C 180,E1 -19954.426,E2 -19954.426} C_VEL
LIN {X 0,Y 227.948,Z 414.716,A -85,B 0,C 180,E1 -19958.286,E2 -19958.286} C_VEL
LIN {X 0,Y 228.036,Z 414.703,A -85,B 0,C 180,E1 -19962.826,E2 -19962.826} C_VEL
LIN {X 0,Y 228.095,Z 414.698,A -85,B 0,C 180,E1 -19967.545,E2 -19967.545} C_VEL
LIN {X 0,Y 228.327,Z 414.669,A -85,B 0,C 180,E1 -19971.147,E2 -19971.147} C_VEL
LIN {X 0,Y 228.36,Z 414.657,A -85,B 0,C 180,E1 -19972.929,E2 -19972.929} C_VEL
LIN {X 0,Y 228.557,Z 414.64,A -85,B 0,C 180,E1 -19978.238,E2 -19978.238} C_VEL
LIN {X 0,Y 228.556,Z 414.64,A -85,B 0,C 180,E1 -19981.762,E2 -19981.762} C_VEL
LIN {X 0,Y 228.36,Z 414.665,A -85,B 0,C 180,E1 -19987.071,E2 -19987.071} C_VEL
LIN {X 0,Y 228.173,Z 414.686,A -85,B 0,C 180,E1 -19990.65,E2 -19990.65} C_VEL
LIN {X 0,Y 228.059,Z 414.701,A -85,B 0,C 180,E1 -19996.102,E2 -19996.102} C_VEL
LIN {X 0,Y 227.944,Z 414.717,A -85,B 0,C 180,E1 -19999.825,E2 -19999.825} C_VEL
LIN {X 0,Y 227.915,Z 414.72,A -85,B 0,C 180,E1 -20003.633,E2 -20003.633} C_VEL
LIN {X 0,Y 227.88,Z 414.725,A -85,B 0,C 180,E1 -20007.556,E2 -20007.556} C_VEL
LIN {X 0,Y 227.87,Z 414.727,A -85,B 0,C 180,E1 -20011.622,E2 -20011.622} C_VEL
LIN {X 0,Y 227.901,Z 414.723,A -85,B 0,C 180,E1 -20015.868,E2 -20015.868} C_VEL
